BEGIN
   BB_G1.Konfig.Res_0 := FALSE;
   BB_G1.Konfig.Res_1 := FALSE;
   BB_G1.Konfig.Res_2 := FALSE;
   BB_G1.Konfig.Res_3 := FALSE;
   BB_G1.Konfig.Res_4 := FALSE;
   BB_G1.Konfig.Res_5 := FALSE;
   BB_G1.Konfig.Res_6 := FALSE;
   BB_G1.Konfig.Res_7 := FALSE;
   BB_G1.Konfig.Res_8 := FALSE;
   BB_G1.Konfig.Res_9 := FALSE;
   BB_G1.Konfig.Res_10 := FALSE;
   BB_G1.Konfig.Res_11 := FALSE;
   BB_G1.Konfig.Res_12 := FALSE;
   BB_G1.Konfig.Res_13 := FALSE;
   BB_G1.Konfig.Res_14 := FALSE;
   BB_G1.Konfig.Res_15 := FALSE;
   BB_G1.Konfig.Res_16 := FALSE;
   BB_G1.Konfig.Res_17 := FALSE;
   BB_G1.Konfig.Res_18 := FALSE;
   BB_G1.Konfig.Res_19 := FALSE;
   BB_G1.Konfig.Res_20 := FALSE;
   BB_G1.Konfig.Res_21 := FALSE;
   BB_G1.Konfig.Res_22 := FALSE;
   BB_G1.Konfig.Res_23 := FALSE;
   BB_G1.Konfig.Res_24 := FALSE;
   BB_G1.Konfig.Res_25 := FALSE;
   BB_G1.Konfig.Res_26 := FALSE;
   BB_G1.Konfig.Res_27 := FALSE;
   BB_G1.Konfig.Res_28 := FALSE;
   BB_G1.Konfig.Res_29 := FALSE;
   BB_G1.Konfig.Res_30 := FALSE;
   BB_G1.Konfig.Prm_Set := FALSE;
   BB_G1.P_nenn := 1.0;
   BB_G1.EZ_max := 0;
   BB_G1.AZ_min := 5;
   BB_G1.AZ_Rev := 10;
   BB_G1.VZ_St := 5;
   BB_G1.UeZ_Endl := 120;
   BB_G1.UeZ_BF := 120;
   BB_G1.Prio_NS := 0;
   BB_G1.Prio_ECS := 0;
   BB_G1.Prio_NA := 0;
   BB_G1.ESV_NA := 5;
   BB_G2.Konfig.Res_0 := FALSE;
   BB_G2.Konfig.Res_1 := FALSE;
   BB_G2.Konfig.Res_2 := FALSE;
   BB_G2.Konfig.Res_3 := FALSE;
   BB_G2.Konfig.Res_4 := FALSE;
   BB_G2.Konfig.Res_5 := FALSE;
   BB_G2.Konfig.Res_6 := FALSE;
   BB_G2.Konfig.Res_7 := FALSE;
   BB_G2.Konfig.Res_8 := FALSE;
   BB_G2.Konfig.Res_9 := FALSE;
   BB_G2.Konfig.Res_10 := FALSE;
   BB_G2.Konfig.Res_11 := FALSE;
   BB_G2.Konfig.Res_12 := FALSE;
   BB_G2.Konfig.Res_13 := FALSE;
   BB_G2.Konfig.Res_14 := FALSE;
   BB_G2.Konfig.Res_15 := FALSE;
   BB_G2.Konfig.Res_16 := FALSE;
   BB_G2.Konfig.Res_17 := FALSE;
   BB_G2.Konfig.Res_18 := FALSE;
   BB_G2.Konfig.Res_19 := FALSE;
   BB_G2.Konfig.Res_20 := FALSE;
   BB_G2.Konfig.Res_21 := FALSE;
   BB_G2.Konfig.Res_22 := FALSE;
   BB_G2.Konfig.Res_23 := FALSE;
   BB_G2.Konfig.Res_24 := FALSE;
   BB_G2.Konfig.Res_25 := FALSE;
   BB_G2.Konfig.Res_26 := FALSE;
   BB_G2.Konfig.Res_27 := FALSE;
   BB_G2.Konfig.Res_28 := FALSE;
   BB_G2.Konfig.Res_29 := FALSE;
   BB_G2.Konfig.Res_30 := FALSE;
   BB_G2.Konfig.Prm_Set := FALSE;
   BB_G2.P_nenn := 1.0;
   BB_G2.EZ_max := 0;
   BB_G2.AZ_min := 5;
   BB_G2.AZ_Rev := 10;
   BB_G2.VZ_St := 5;
   BB_G2.UeZ_Endl := 120;
   BB_G2.UeZ_BF := 15;
   BB_G2.Prio_NS := 0;
   BB_G2.Prio_ECS := 0;
   BB_G2.Prio_NA := 0;
   BB_G2.ESV_NA := 5;
   BB_G3.Konfig.Res_0 := FALSE;
   BB_G3.Konfig.Res_1 := FALSE;
   BB_G3.Konfig.Res_2 := FALSE;
   BB_G3.Konfig.Res_3 := FALSE;
   BB_G3.Konfig.Res_4 := FALSE;
   BB_G3.Konfig.Res_5 := FALSE;
   BB_G3.Konfig.Res_6 := FALSE;
   BB_G3.Konfig.Res_7 := FALSE;
   BB_G3.Konfig.Res_8 := FALSE;
   BB_G3.Konfig.Res_9 := FALSE;
   BB_G3.Konfig.Res_10 := FALSE;
   BB_G3.Konfig.Res_11 := FALSE;
   BB_G3.Konfig.Res_12 := FALSE;
   BB_G3.Konfig.Res_13 := FALSE;
   BB_G3.Konfig.Res_14 := FALSE;
   BB_G3.Konfig.Res_15 := FALSE;
   BB_G3.Konfig.Res_16 := FALSE;
   BB_G3.Konfig.Res_17 := FALSE;
   BB_G3.Konfig.Res_18 := FALSE;
   BB_G3.Konfig.Res_19 := FALSE;
   BB_G3.Konfig.Res_20 := FALSE;
   BB_G3.Konfig.Res_21 := FALSE;
   BB_G3.Konfig.Res_22 := FALSE;
   BB_G3.Konfig.Res_23 := FALSE;
   BB_G3.Konfig.Res_24 := FALSE;
   BB_G3.Konfig.Res_25 := FALSE;
   BB_G3.Konfig.Res_26 := FALSE;
   BB_G3.Konfig.Res_27 := FALSE;
   BB_G3.Konfig.Res_28 := FALSE;
   BB_G3.Konfig.Res_29 := FALSE;
   BB_G3.Konfig.Res_30 := FALSE;
   BB_G3.Konfig.Prm_Set := FALSE;
   BB_G3.P_nenn := 1.0;
   BB_G3.EZ_max := 0;
   BB_G3.AZ_min := 5;
   BB_G3.AZ_Rev := 10;
   BB_G3.VZ_St := 5;
   BB_G3.UeZ_Endl := 120;
   BB_G3.UeZ_BF := 15;
   BB_G3.Prio_NS := 0;
   BB_G3.Prio_ECS := 0;
   BB_G3.Prio_NA := 0;
   BB_G3.ESV_NA := 5;
   BB_SHL_G1.Konfig.Res_0 := FALSE;
   BB_SHL_G1.Konfig.Res_1 := FALSE;
   BB_SHL_G1.Konfig.Res_2 := FALSE;
   BB_SHL_G1.Konfig.Res_3 := FALSE;
   BB_SHL_G1.Konfig.Res_4 := FALSE;
   BB_SHL_G1.Konfig.Res_5 := FALSE;
   BB_SHL_G1.Konfig.Res_6 := FALSE;
   BB_SHL_G1.Konfig.Res_7 := FALSE;
   BB_SHL_G1.Konfig.Res_8 := FALSE;
   BB_SHL_G1.Konfig.Res_9 := FALSE;
   BB_SHL_G1.Konfig.Res_10 := FALSE;
   BB_SHL_G1.Konfig.Res_11 := FALSE;
   BB_SHL_G1.Konfig.Res_12 := FALSE;
   BB_SHL_G1.Konfig.Res_13 := FALSE;
   BB_SHL_G1.Konfig.Res_14 := FALSE;
   BB_SHL_G1.Konfig.Res_15 := FALSE;
   BB_SHL_G1.Konfig.Res_16 := FALSE;
   BB_SHL_G1.Konfig.Res_17 := FALSE;
   BB_SHL_G1.Konfig.Res_18 := FALSE;
   BB_SHL_G1.Konfig.Res_19 := FALSE;
   BB_SHL_G1.Konfig.Res_20 := FALSE;
   BB_SHL_G1.Konfig.Res_21 := FALSE;
   BB_SHL_G1.Konfig.Res_22 := FALSE;
   BB_SHL_G1.Konfig.Res_23 := FALSE;
   BB_SHL_G1.Konfig.Res_24 := FALSE;
   BB_SHL_G1.Konfig.Res_25 := FALSE;
   BB_SHL_G1.Konfig.Res_26 := FALSE;
   BB_SHL_G1.Konfig.Res_27 := FALSE;
   BB_SHL_G1.Konfig.Res_28 := FALSE;
   BB_SHL_G1.Konfig.Res_29 := FALSE;
   BB_SHL_G1.Konfig.Res_30 := FALSE;
   BB_SHL_G1.Konfig.Prm_Set := FALSE;
   BB_SHL_G1.P_nenn := 1.0;
   BB_SHL_G1.EZ_max := 0;
   BB_SHL_G1.AZ_min := 5;
   BB_SHL_G1.AZ_Rev := 10;
   BB_SHL_G1.VZ_St := 5;
   BB_SHL_G1.UeZ_Endl := 120;
   BB_SHL_G1.UeZ_BF := 15;
   BB_SHL_G1.Prio_NS := 0;
   BB_SHL_G1.Prio_ECS := 0;
   BB_SHL_G1.Prio_NA := 0;
   BB_SHL_G1.ESV_NA := 5;
   BB_SHL_G2.Konfig.Res_0 := FALSE;
   BB_SHL_G2.Konfig.Res_1 := FALSE;
   BB_SHL_G2.Konfig.Res_2 := FALSE;
   BB_SHL_G2.Konfig.Res_3 := FALSE;
   BB_SHL_G2.Konfig.Res_4 := FALSE;
   BB_SHL_G2.Konfig.Res_5 := FALSE;
   BB_SHL_G2.Konfig.Res_6 := FALSE;
   BB_SHL_G2.Konfig.Res_7 := FALSE;
   BB_SHL_G2.Konfig.Res_8 := FALSE;
   BB_SHL_G2.Konfig.Res_9 := FALSE;
   BB_SHL_G2.Konfig.Res_10 := FALSE;
   BB_SHL_G2.Konfig.Res_11 := FALSE;
   BB_SHL_G2.Konfig.Res_12 := FALSE;
   BB_SHL_G2.Konfig.Res_13 := FALSE;
   BB_SHL_G2.Konfig.Res_14 := FALSE;
   BB_SHL_G2.Konfig.Res_15 := FALSE;
   BB_SHL_G2.Konfig.Res_16 := FALSE;
   BB_SHL_G2.Konfig.Res_17 := FALSE;
   BB_SHL_G2.Konfig.Res_18 := FALSE;
   BB_SHL_G2.Konfig.Res_19 := FALSE;
   BB_SHL_G2.Konfig.Res_20 := FALSE;
   BB_SHL_G2.Konfig.Res_21 := FALSE;
   BB_SHL_G2.Konfig.Res_22 := FALSE;
   BB_SHL_G2.Konfig.Res_23 := FALSE;
   BB_SHL_G2.Konfig.Res_24 := FALSE;
   BB_SHL_G2.Konfig.Res_25 := FALSE;
   BB_SHL_G2.Konfig.Res_26 := FALSE;
   BB_SHL_G2.Konfig.Res_27 := FALSE;
   BB_SHL_G2.Konfig.Res_28 := FALSE;
   BB_SHL_G2.Konfig.Res_29 := FALSE;
   BB_SHL_G2.Konfig.Res_30 := FALSE;
   BB_SHL_G2.Konfig.Prm_Set := FALSE;
   BB_SHL_G2.P_nenn := 1.0;
   BB_SHL_G2.EZ_max := 0;
   BB_SHL_G2.AZ_min := 5;
   BB_SHL_G2.AZ_Rev := 10;
   BB_SHL_G2.VZ_St := 5;
   BB_SHL_G2.UeZ_Endl := 120;
   BB_SHL_G2.UeZ_BF := 15;
   BB_SHL_G2.Prio_NS := 0;
   BB_SHL_G2.Prio_ECS := 0;
   BB_SHL_G2.Prio_NA := 0;
   BB_SHL_G2.ESV_NA := 5;
   BB_SHL_G3.Konfig.Res_0 := FALSE;
   BB_SHL_G3.Konfig.Res_1 := FALSE;
   BB_SHL_G3.Konfig.Res_2 := FALSE;
   BB_SHL_G3.Konfig.Res_3 := FALSE;
   BB_SHL_G3.Konfig.Res_4 := FALSE;
   BB_SHL_G3.Konfig.Res_5 := FALSE;
   BB_SHL_G3.Konfig.Res_6 := FALSE;
   BB_SHL_G3.Konfig.Res_7 := FALSE;
   BB_SHL_G3.Konfig.Res_8 := FALSE;
   BB_SHL_G3.Konfig.Res_9 := FALSE;
   BB_SHL_G3.Konfig.Res_10 := FALSE;
   BB_SHL_G3.Konfig.Res_11 := FALSE;
   BB_SHL_G3.Konfig.Res_12 := FALSE;
   BB_SHL_G3.Konfig.Res_13 := FALSE;
   BB_SHL_G3.Konfig.Res_14 := FALSE;
   BB_SHL_G3.Konfig.Res_15 := FALSE;
   BB_SHL_G3.Konfig.Res_16 := FALSE;
   BB_SHL_G3.Konfig.Res_17 := FALSE;
   BB_SHL_G3.Konfig.Res_18 := FALSE;
   BB_SHL_G3.Konfig.Res_19 := FALSE;
   BB_SHL_G3.Konfig.Res_20 := FALSE;
   BB_SHL_G3.Konfig.Res_21 := FALSE;
   BB_SHL_G3.Konfig.Res_22 := FALSE;
   BB_SHL_G3.Konfig.Res_23 := FALSE;
   BB_SHL_G3.Konfig.Res_24 := FALSE;
   BB_SHL_G3.Konfig.Res_25 := FALSE;
   BB_SHL_G3.Konfig.Res_26 := FALSE;
   BB_SHL_G3.Konfig.Res_27 := FALSE;
   BB_SHL_G3.Konfig.Res_28 := FALSE;
   BB_SHL_G3.Konfig.Res_29 := FALSE;
   BB_SHL_G3.Konfig.Res_30 := FALSE;
   BB_SHL_G3.Konfig.Prm_Set := FALSE;
   BB_SHL_G3.P_nenn := 1.0;
   BB_SHL_G3.EZ_max := 0;
   BB_SHL_G3.AZ_min := 5;
   BB_SHL_G3.AZ_Rev := 10;
   BB_SHL_G3.VZ_St := 5;
   BB_SHL_G3.UeZ_Endl := 120;
   BB_SHL_G3.UeZ_BF := 15;
   BB_SHL_G3.Prio_NS := 0;
   BB_SHL_G3.Prio_ECS := 0;
   BB_SHL_G3.Prio_NA := 0;
   BB_SHL_G3.ESV_NA := 5;
   BB_AV.Konfig.Res_0 := FALSE;
   BB_AV.Konfig.Res_1 := FALSE;
   BB_AV.Konfig.Res_2 := FALSE;
   BB_AV.Konfig.Res_3 := FALSE;
   BB_AV.Konfig.Res_4 := FALSE;
   BB_AV.Konfig.Res_5 := FALSE;
   BB_AV.Konfig.Res_6 := FALSE;
   BB_AV.Konfig.Res_7 := FALSE;
   BB_AV.Konfig.Res_8 := FALSE;
   BB_AV.Konfig.Res_9 := FALSE;
   BB_AV.Konfig.Res_10 := FALSE;
   BB_AV.Konfig.Res_11 := FALSE;
   BB_AV.Konfig.Res_12 := FALSE;
   BB_AV.Konfig.Res_13 := FALSE;
   BB_AV.Konfig.Res_14 := FALSE;
   BB_AV.Konfig.Res_15 := FALSE;
   BB_AV.Konfig.Res_16 := FALSE;
   BB_AV.Konfig.Res_17 := FALSE;
   BB_AV.Konfig.Res_18 := FALSE;
   BB_AV.Konfig.Res_19 := FALSE;
   BB_AV.Konfig.Res_20 := FALSE;
   BB_AV.Konfig.Res_21 := FALSE;
   BB_AV.Konfig.Res_22 := FALSE;
   BB_AV.Konfig.Res_23 := FALSE;
   BB_AV.Konfig.Res_24 := FALSE;
   BB_AV.Konfig.Res_25 := FALSE;
   BB_AV.Konfig.Res_26 := FALSE;
   BB_AV.Konfig.Res_27 := FALSE;
   BB_AV.Konfig.Res_28 := FALSE;
   BB_AV.Konfig.Res_29 := FALSE;
   BB_AV.Konfig.Res_30 := FALSE;
   BB_AV.Konfig.Prm_Set := FALSE;
   BB_AV.P_nenn := 1.0;
   BB_AV.EZ_max := 0;
   BB_AV.AZ_min := 5;
   BB_AV.AZ_Rev := 10;
   BB_AV.VZ_St := 5;
   BB_AV.UeZ_Endl := 120;
   BB_AV.UeZ_BF := 15;
   BB_AV.Prio_NS := 0;
   BB_AV.Prio_ECS := 0;
   BB_AV.Prio_NA := 0;
   BB_AV.ESV_NA := 5;
   BB_LS1.Konfig.Res_0 := FALSE;
   BB_LS1.Konfig.Res_1 := FALSE;
   BB_LS1.Konfig.Res_2 := FALSE;
   BB_LS1.Konfig.Res_3 := FALSE;
   BB_LS1.Konfig.Res_4 := FALSE;
   BB_LS1.Konfig.Res_5 := FALSE;
   BB_LS1.Konfig.Res_6 := FALSE;
   BB_LS1.Konfig.Res_7 := FALSE;
   BB_LS1.Konfig.Res_8 := FALSE;
   BB_LS1.Konfig.Res_9 := FALSE;
   BB_LS1.Konfig.Res_10 := FALSE;
   BB_LS1.Konfig.Res_11 := FALSE;
   BB_LS1.Konfig.Res_12 := FALSE;
   BB_LS1.Konfig.Res_13 := FALSE;
   BB_LS1.Konfig.Res_14 := FALSE;
   BB_LS1.Konfig.Res_15 := FALSE;
   BB_LS1.Konfig.Res_16 := FALSE;
   BB_LS1.Konfig.Res_17 := FALSE;
   BB_LS1.Konfig.Res_18 := FALSE;
   BB_LS1.Konfig.Res_19 := FALSE;
   BB_LS1.Konfig.Res_20 := FALSE;
   BB_LS1.Konfig.Res_21 := FALSE;
   BB_LS1.Konfig.Res_22 := FALSE;
   BB_LS1.Konfig.Res_23 := FALSE;
   BB_LS1.Konfig.Res_24 := FALSE;
   BB_LS1.Konfig.Res_25 := FALSE;
   BB_LS1.Konfig.Res_26 := FALSE;
   BB_LS1.Konfig.Res_27 := FALSE;
   BB_LS1.Konfig.Res_28 := FALSE;
   BB_LS1.Konfig.Res_29 := FALSE;
   BB_LS1.Konfig.Res_30 := FALSE;
   BB_LS1.Konfig.Prm_Set := FALSE;
   BB_LS1.P_nenn := 1.0;
   BB_LS1.EZ_max := 0;
   BB_LS1.AZ_min := 5;
   BB_LS1.AZ_Rev := 10;
   BB_LS1.VZ_St := 5;
   BB_LS1.UeZ_Endl := 120;
   BB_LS1.UeZ_BF := 15;
   BB_LS1.Prio_NS := 0;
   BB_LS1.Prio_ECS := 0;
   BB_LS1.Prio_NA := 0;
   BB_LS1.ESV_NA := 5;
   BB_LS2.Konfig.Res_0 := FALSE;
   BB_LS2.Konfig.Res_1 := FALSE;
   BB_LS2.Konfig.Res_2 := FALSE;
   BB_LS2.Konfig.Res_3 := FALSE;
   BB_LS2.Konfig.Res_4 := FALSE;
   BB_LS2.Konfig.Res_5 := FALSE;
   BB_LS2.Konfig.Res_6 := FALSE;
   BB_LS2.Konfig.Res_7 := FALSE;
   BB_LS2.Konfig.Res_8 := FALSE;
   BB_LS2.Konfig.Res_9 := FALSE;
   BB_LS2.Konfig.Res_10 := FALSE;
   BB_LS2.Konfig.Res_11 := FALSE;
   BB_LS2.Konfig.Res_12 := FALSE;
   BB_LS2.Konfig.Res_13 := FALSE;
   BB_LS2.Konfig.Res_14 := FALSE;
   BB_LS2.Konfig.Res_15 := FALSE;
   BB_LS2.Konfig.Res_16 := FALSE;
   BB_LS2.Konfig.Res_17 := FALSE;
   BB_LS2.Konfig.Res_18 := FALSE;
   BB_LS2.Konfig.Res_19 := FALSE;
   BB_LS2.Konfig.Res_20 := FALSE;
   BB_LS2.Konfig.Res_21 := FALSE;
   BB_LS2.Konfig.Res_22 := FALSE;
   BB_LS2.Konfig.Res_23 := FALSE;
   BB_LS2.Konfig.Res_24 := FALSE;
   BB_LS2.Konfig.Res_25 := FALSE;
   BB_LS2.Konfig.Res_26 := FALSE;
   BB_LS2.Konfig.Res_27 := FALSE;
   BB_LS2.Konfig.Res_28 := FALSE;
   BB_LS2.Konfig.Res_29 := FALSE;
   BB_LS2.Konfig.Res_30 := FALSE;
   BB_LS2.Konfig.Prm_Set := FALSE;
   BB_LS2.P_nenn := 1.0;
   BB_LS2.EZ_max := 0;
   BB_LS2.AZ_min := 5;
   BB_LS2.AZ_Rev := 10;
   BB_LS2.VZ_St := 5;
   BB_LS2.UeZ_Endl := 120;
   BB_LS2.UeZ_BF := 15;
   BB_LS2.Prio_NS := 0;
   BB_LS2.Prio_ECS := 0;
   BB_LS2.Prio_NA := 0;
   BB_LS2.ESV_NA := 5;
   BB1_RZP1.Konfig.Res_0 := FALSE;
   BB1_RZP1.Konfig.Res_1 := FALSE;
   BB1_RZP1.Konfig.Res_2 := FALSE;
   BB1_RZP1.Konfig.Res_3 := FALSE;
   BB1_RZP1.Konfig.Res_4 := FALSE;
   BB1_RZP1.Konfig.Res_5 := FALSE;
   BB1_RZP1.Konfig.Res_6 := FALSE;
   BB1_RZP1.Konfig.Res_7 := FALSE;
   BB1_RZP1.Konfig.Res_8 := FALSE;
   BB1_RZP1.Konfig.Res_9 := FALSE;
   BB1_RZP1.Konfig.Res_10 := FALSE;
   BB1_RZP1.Konfig.Res_11 := FALSE;
   BB1_RZP1.Konfig.Res_12 := FALSE;
   BB1_RZP1.Konfig.Res_13 := FALSE;
   BB1_RZP1.Konfig.Res_14 := FALSE;
   BB1_RZP1.Konfig.Res_15 := FALSE;
   BB1_RZP1.Konfig.Res_16 := FALSE;
   BB1_RZP1.Konfig.Res_17 := FALSE;
   BB1_RZP1.Konfig.Res_18 := FALSE;
   BB1_RZP1.Konfig.Res_19 := FALSE;
   BB1_RZP1.Konfig.Res_20 := FALSE;
   BB1_RZP1.Konfig.Res_21 := FALSE;
   BB1_RZP1.Konfig.Res_22 := FALSE;
   BB1_RZP1.Konfig.Res_23 := FALSE;
   BB1_RZP1.Konfig.Res_24 := FALSE;
   BB1_RZP1.Konfig.Res_25 := FALSE;
   BB1_RZP1.Konfig.Res_26 := FALSE;
   BB1_RZP1.Konfig.Res_27 := FALSE;
   BB1_RZP1.Konfig.Res_28 := FALSE;
   BB1_RZP1.Konfig.Res_29 := FALSE;
   BB1_RZP1.Konfig.Res_30 := FALSE;
   BB1_RZP1.Konfig.Prm_Set := FALSE;
   BB1_RZP1.P_nenn := 2.0;
   BB1_RZP1.EZ_max := 0;
   BB1_RZP1.AZ_min := 5;
   BB1_RZP1.AZ_Rev := 10;
   BB1_RZP1.VZ_St := 5;
   BB1_RZP1.UeZ_Endl := 300;
   BB1_RZP1.UeZ_BF := 15;
   BB1_RZP1.Prio_NS := 0;
   BB1_RZP1.Prio_ECS := 0;
   BB1_RZP1.Prio_NA := 0;
   BB1_RZP1.ESV_NA := 5;
   BB1_RZP2.Konfig.Res_0 := FALSE;
   BB1_RZP2.Konfig.Res_1 := FALSE;
   BB1_RZP2.Konfig.Res_2 := FALSE;
   BB1_RZP2.Konfig.Res_3 := FALSE;
   BB1_RZP2.Konfig.Res_4 := FALSE;
   BB1_RZP2.Konfig.Res_5 := FALSE;
   BB1_RZP2.Konfig.Res_6 := FALSE;
   BB1_RZP2.Konfig.Res_7 := FALSE;
   BB1_RZP2.Konfig.Res_8 := FALSE;
   BB1_RZP2.Konfig.Res_9 := FALSE;
   BB1_RZP2.Konfig.Res_10 := FALSE;
   BB1_RZP2.Konfig.Res_11 := FALSE;
   BB1_RZP2.Konfig.Res_12 := FALSE;
   BB1_RZP2.Konfig.Res_13 := FALSE;
   BB1_RZP2.Konfig.Res_14 := FALSE;
   BB1_RZP2.Konfig.Res_15 := FALSE;
   BB1_RZP2.Konfig.Res_16 := FALSE;
   BB1_RZP2.Konfig.Res_17 := FALSE;
   BB1_RZP2.Konfig.Res_18 := FALSE;
   BB1_RZP2.Konfig.Res_19 := FALSE;
   BB1_RZP2.Konfig.Res_20 := FALSE;
   BB1_RZP2.Konfig.Res_21 := FALSE;
   BB1_RZP2.Konfig.Res_22 := FALSE;
   BB1_RZP2.Konfig.Res_23 := FALSE;
   BB1_RZP2.Konfig.Res_24 := FALSE;
   BB1_RZP2.Konfig.Res_25 := FALSE;
   BB1_RZP2.Konfig.Res_26 := FALSE;
   BB1_RZP2.Konfig.Res_27 := FALSE;
   BB1_RZP2.Konfig.Res_28 := FALSE;
   BB1_RZP2.Konfig.Res_29 := FALSE;
   BB1_RZP2.Konfig.Res_30 := FALSE;
   BB1_RZP2.Konfig.Prm_Set := FALSE;
   BB1_RZP2.P_nenn := 1.0;
   BB1_RZP2.EZ_max := 0;
   BB1_RZP2.AZ_min := 5;
   BB1_RZP2.AZ_Rev := 10;
   BB1_RZP2.VZ_St := 5;
   BB1_RZP2.UeZ_Endl := 120;
   BB1_RZP2.UeZ_BF := 15;
   BB1_RZP2.Prio_NS := 0;
   BB1_RZP2.Prio_ECS := 0;
   BB1_RZP2.Prio_NA := 0;
   BB1_RZP2.ESV_NA := 5;
   BB1_UeSP.Konfig.Res_0 := FALSE;
   BB1_UeSP.Konfig.Res_1 := FALSE;
   BB1_UeSP.Konfig.Res_2 := FALSE;
   BB1_UeSP.Konfig.Res_3 := FALSE;
   BB1_UeSP.Konfig.Res_4 := FALSE;
   BB1_UeSP.Konfig.Res_5 := FALSE;
   BB1_UeSP.Konfig.Res_6 := FALSE;
   BB1_UeSP.Konfig.Res_7 := FALSE;
   BB1_UeSP.Konfig.Res_8 := FALSE;
   BB1_UeSP.Konfig.Res_9 := FALSE;
   BB1_UeSP.Konfig.Res_10 := FALSE;
   BB1_UeSP.Konfig.Res_11 := FALSE;
   BB1_UeSP.Konfig.Res_12 := FALSE;
   BB1_UeSP.Konfig.Res_13 := FALSE;
   BB1_UeSP.Konfig.Res_14 := FALSE;
   BB1_UeSP.Konfig.Res_15 := FALSE;
   BB1_UeSP.Konfig.Res_16 := FALSE;
   BB1_UeSP.Konfig.Res_17 := FALSE;
   BB1_UeSP.Konfig.Res_18 := FALSE;
   BB1_UeSP.Konfig.Res_19 := FALSE;
   BB1_UeSP.Konfig.Res_20 := FALSE;
   BB1_UeSP.Konfig.Res_21 := FALSE;
   BB1_UeSP.Konfig.Res_22 := FALSE;
   BB1_UeSP.Konfig.Res_23 := FALSE;
   BB1_UeSP.Konfig.Res_24 := FALSE;
   BB1_UeSP.Konfig.Res_25 := FALSE;
   BB1_UeSP.Konfig.Res_26 := FALSE;
   BB1_UeSP.Konfig.Res_27 := FALSE;
   BB1_UeSP.Konfig.Res_28 := FALSE;
   BB1_UeSP.Konfig.Res_29 := FALSE;
   BB1_UeSP.Konfig.Res_30 := FALSE;
   BB1_UeSP.Konfig.Prm_Set := FALSE;
   BB1_UeSP.P_nenn := 1.0;
   BB1_UeSP.EZ_max := 0;
   BB1_UeSP.AZ_min := 5;
   BB1_UeSP.AZ_Rev := 10;
   BB1_UeSP.VZ_St := 5;
   BB1_UeSP.UeZ_Endl := 120;
   BB1_UeSP.UeZ_BF := 15;
   BB1_UeSP.Prio_NS := 0;
   BB1_UeSP.Prio_ECS := 0;
   BB1_UeSP.Prio_NA := 0;
   BB1_UeSP.ESV_NA := 5;
   BB1_AS1.Konfig.Res_0 := FALSE;
   BB1_AS1.Konfig.Res_1 := FALSE;
   BB1_AS1.Konfig.Res_2 := FALSE;
   BB1_AS1.Konfig.Res_3 := FALSE;
   BB1_AS1.Konfig.Res_4 := FALSE;
   BB1_AS1.Konfig.Res_5 := FALSE;
   BB1_AS1.Konfig.Res_6 := FALSE;
   BB1_AS1.Konfig.Res_7 := FALSE;
   BB1_AS1.Konfig.Res_8 := FALSE;
   BB1_AS1.Konfig.Res_9 := FALSE;
   BB1_AS1.Konfig.Res_10 := FALSE;
   BB1_AS1.Konfig.Res_11 := FALSE;
   BB1_AS1.Konfig.Res_12 := FALSE;
   BB1_AS1.Konfig.Res_13 := FALSE;
   BB1_AS1.Konfig.Res_14 := FALSE;
   BB1_AS1.Konfig.Res_15 := FALSE;
   BB1_AS1.Konfig.Res_16 := FALSE;
   BB1_AS1.Konfig.Res_17 := FALSE;
   BB1_AS1.Konfig.Res_18 := FALSE;
   BB1_AS1.Konfig.Res_19 := FALSE;
   BB1_AS1.Konfig.Res_20 := FALSE;
   BB1_AS1.Konfig.Res_21 := FALSE;
   BB1_AS1.Konfig.Res_22 := FALSE;
   BB1_AS1.Konfig.Res_23 := FALSE;
   BB1_AS1.Konfig.Res_24 := FALSE;
   BB1_AS1.Konfig.Res_25 := FALSE;
   BB1_AS1.Konfig.Res_26 := FALSE;
   BB1_AS1.Konfig.Res_27 := FALSE;
   BB1_AS1.Konfig.Res_28 := FALSE;
   BB1_AS1.Konfig.Res_29 := FALSE;
   BB1_AS1.Konfig.Res_30 := FALSE;
   BB1_AS1.Konfig.Prm_Set := FALSE;
   BB1_AS1.P_nenn := 1.0;
   BB1_AS1.EZ_max := 0;
   BB1_AS1.AZ_min := 5;
   BB1_AS1.AZ_Rev := 10;
   BB1_AS1.VZ_St := 5;
   BB1_AS1.UeZ_Endl := 120;
   BB1_AS1.UeZ_BF := 15;
   BB1_AS1.Prio_NS := 0;
   BB1_AS1.Prio_ECS := 0;
   BB1_AS1.Prio_NA := 0;
   BB1_AS1.ESV_NA := 5;
   BB1_AS2.Konfig.Res_0 := FALSE;
   BB1_AS2.Konfig.Res_1 := FALSE;
   BB1_AS2.Konfig.Res_2 := FALSE;
   BB1_AS2.Konfig.Res_3 := FALSE;
   BB1_AS2.Konfig.Res_4 := FALSE;
   BB1_AS2.Konfig.Res_5 := FALSE;
   BB1_AS2.Konfig.Res_6 := FALSE;
   BB1_AS2.Konfig.Res_7 := FALSE;
   BB1_AS2.Konfig.Res_8 := FALSE;
   BB1_AS2.Konfig.Res_9 := FALSE;
   BB1_AS2.Konfig.Res_10 := FALSE;
   BB1_AS2.Konfig.Res_11 := FALSE;
   BB1_AS2.Konfig.Res_12 := FALSE;
   BB1_AS2.Konfig.Res_13 := FALSE;
   BB1_AS2.Konfig.Res_14 := FALSE;
   BB1_AS2.Konfig.Res_15 := FALSE;
   BB1_AS2.Konfig.Res_16 := FALSE;
   BB1_AS2.Konfig.Res_17 := FALSE;
   BB1_AS2.Konfig.Res_18 := FALSE;
   BB1_AS2.Konfig.Res_19 := FALSE;
   BB1_AS2.Konfig.Res_20 := FALSE;
   BB1_AS2.Konfig.Res_21 := FALSE;
   BB1_AS2.Konfig.Res_22 := FALSE;
   BB1_AS2.Konfig.Res_23 := FALSE;
   BB1_AS2.Konfig.Res_24 := FALSE;
   BB1_AS2.Konfig.Res_25 := FALSE;
   BB1_AS2.Konfig.Res_26 := FALSE;
   BB1_AS2.Konfig.Res_27 := FALSE;
   BB1_AS2.Konfig.Res_28 := FALSE;
   BB1_AS2.Konfig.Res_29 := FALSE;
   BB1_AS2.Konfig.Res_30 := FALSE;
   BB1_AS2.Konfig.Prm_Set := FALSE;
   BB1_AS2.P_nenn := 1.0;
   BB1_AS2.EZ_max := 0;
   BB1_AS2.AZ_min := 5;
   BB1_AS2.AZ_Rev := 10;
   BB1_AS2.VZ_St := 5;
   BB1_AS2.UeZ_Endl := 120;
   BB1_AS2.UeZ_BF := 15;
   BB1_AS2.Prio_NS := 0;
   BB1_AS2.Prio_ECS := 0;
   BB1_AS2.Prio_NA := 0;
   BB1_AS2.ESV_NA := 5;
   BB1_SR1.Konfig.Res_0 := FALSE;
   BB1_SR1.Konfig.Res_1 := FALSE;
   BB1_SR1.Konfig.Res_2 := FALSE;
   BB1_SR1.Konfig.Res_3 := FALSE;
   BB1_SR1.Konfig.Res_4 := FALSE;
   BB1_SR1.Konfig.Res_5 := FALSE;
   BB1_SR1.Konfig.Res_6 := FALSE;
   BB1_SR1.Konfig.Res_7 := FALSE;
   BB1_SR1.Konfig.Res_8 := FALSE;
   BB1_SR1.Konfig.Res_9 := FALSE;
   BB1_SR1.Konfig.Res_10 := FALSE;
   BB1_SR1.Konfig.Res_11 := FALSE;
   BB1_SR1.Konfig.Res_12 := FALSE;
   BB1_SR1.Konfig.Res_13 := FALSE;
   BB1_SR1.Konfig.Res_14 := FALSE;
   BB1_SR1.Konfig.Res_15 := FALSE;
   BB1_SR1.Konfig.Res_16 := FALSE;
   BB1_SR1.Konfig.Res_17 := FALSE;
   BB1_SR1.Konfig.Res_18 := FALSE;
   BB1_SR1.Konfig.Res_19 := FALSE;
   BB1_SR1.Konfig.Res_20 := FALSE;
   BB1_SR1.Konfig.Res_21 := FALSE;
   BB1_SR1.Konfig.Res_22 := FALSE;
   BB1_SR1.Konfig.Res_23 := FALSE;
   BB1_SR1.Konfig.Res_24 := FALSE;
   BB1_SR1.Konfig.Res_25 := FALSE;
   BB1_SR1.Konfig.Res_26 := FALSE;
   BB1_SR1.Konfig.Res_27 := FALSE;
   BB1_SR1.Konfig.Res_28 := FALSE;
   BB1_SR1.Konfig.Res_29 := FALSE;
   BB1_SR1.Konfig.Res_30 := FALSE;
   BB1_SR1.Konfig.Prm_Set := FALSE;
   BB1_SR1.P_nenn := 1.0;
   BB1_SR1.EZ_max := 0;
   BB1_SR1.AZ_min := 5;
   BB1_SR1.AZ_Rev := 10;
   BB1_SR1.VZ_St := 5;
   BB1_SR1.UeZ_Endl := 120;
   BB1_SR1.UeZ_BF := 15;
   BB1_SR1.Prio_NS := 0;
   BB1_SR1.Prio_ECS := 0;
   BB1_SR1.Prio_NA := 0;
   BB1_SR1.ESV_NA := 5;
   BB1_SR2.Konfig.Res_0 := FALSE;
   BB1_SR2.Konfig.Res_1 := FALSE;
   BB1_SR2.Konfig.Res_2 := FALSE;
   BB1_SR2.Konfig.Res_3 := FALSE;
   BB1_SR2.Konfig.Res_4 := FALSE;
   BB1_SR2.Konfig.Res_5 := FALSE;
   BB1_SR2.Konfig.Res_6 := FALSE;
   BB1_SR2.Konfig.Res_7 := FALSE;
   BB1_SR2.Konfig.Res_8 := FALSE;
   BB1_SR2.Konfig.Res_9 := FALSE;
   BB1_SR2.Konfig.Res_10 := FALSE;
   BB1_SR2.Konfig.Res_11 := FALSE;
   BB1_SR2.Konfig.Res_12 := FALSE;
   BB1_SR2.Konfig.Res_13 := FALSE;
   BB1_SR2.Konfig.Res_14 := FALSE;
   BB1_SR2.Konfig.Res_15 := FALSE;
   BB1_SR2.Konfig.Res_16 := FALSE;
   BB1_SR2.Konfig.Res_17 := FALSE;
   BB1_SR2.Konfig.Res_18 := FALSE;
   BB1_SR2.Konfig.Res_19 := FALSE;
   BB1_SR2.Konfig.Res_20 := FALSE;
   BB1_SR2.Konfig.Res_21 := FALSE;
   BB1_SR2.Konfig.Res_22 := FALSE;
   BB1_SR2.Konfig.Res_23 := FALSE;
   BB1_SR2.Konfig.Res_24 := FALSE;
   BB1_SR2.Konfig.Res_25 := FALSE;
   BB1_SR2.Konfig.Res_26 := FALSE;
   BB1_SR2.Konfig.Res_27 := FALSE;
   BB1_SR2.Konfig.Res_28 := FALSE;
   BB1_SR2.Konfig.Res_29 := FALSE;
   BB1_SR2.Konfig.Res_30 := FALSE;
   BB1_SR2.Konfig.Prm_Set := FALSE;
   BB1_SR2.P_nenn := 1.0;
   BB1_SR2.EZ_max := 0;
   BB1_SR2.AZ_min := 5;
   BB1_SR2.AZ_Rev := 10;
   BB1_SR2.VZ_St := 5;
   BB1_SR2.UeZ_Endl := 120;
   BB1_SR2.UeZ_BF := 15;
   BB1_SR2.Prio_NS := 0;
   BB1_SR2.Prio_ECS := 0;
   BB1_SR2.Prio_NA := 0;
   BB1_SR2.ESV_NA := 5;
   BB2_RZP1.Konfig.Res_0 := FALSE;
   BB2_RZP1.Konfig.Res_1 := FALSE;
   BB2_RZP1.Konfig.Res_2 := FALSE;
   BB2_RZP1.Konfig.Res_3 := FALSE;
   BB2_RZP1.Konfig.Res_4 := FALSE;
   BB2_RZP1.Konfig.Res_5 := FALSE;
   BB2_RZP1.Konfig.Res_6 := FALSE;
   BB2_RZP1.Konfig.Res_7 := FALSE;
   BB2_RZP1.Konfig.Res_8 := FALSE;
   BB2_RZP1.Konfig.Res_9 := FALSE;
   BB2_RZP1.Konfig.Res_10 := FALSE;
   BB2_RZP1.Konfig.Res_11 := FALSE;
   BB2_RZP1.Konfig.Res_12 := FALSE;
   BB2_RZP1.Konfig.Res_13 := FALSE;
   BB2_RZP1.Konfig.Res_14 := FALSE;
   BB2_RZP1.Konfig.Res_15 := FALSE;
   BB2_RZP1.Konfig.Res_16 := FALSE;
   BB2_RZP1.Konfig.Res_17 := FALSE;
   BB2_RZP1.Konfig.Res_18 := FALSE;
   BB2_RZP1.Konfig.Res_19 := FALSE;
   BB2_RZP1.Konfig.Res_20 := FALSE;
   BB2_RZP1.Konfig.Res_21 := FALSE;
   BB2_RZP1.Konfig.Res_22 := FALSE;
   BB2_RZP1.Konfig.Res_23 := FALSE;
   BB2_RZP1.Konfig.Res_24 := FALSE;
   BB2_RZP1.Konfig.Res_25 := FALSE;
   BB2_RZP1.Konfig.Res_26 := FALSE;
   BB2_RZP1.Konfig.Res_27 := FALSE;
   BB2_RZP1.Konfig.Res_28 := FALSE;
   BB2_RZP1.Konfig.Res_29 := FALSE;
   BB2_RZP1.Konfig.Res_30 := FALSE;
   BB2_RZP1.Konfig.Prm_Set := FALSE;
   BB2_RZP1.P_nenn := 1.0;
   BB2_RZP1.EZ_max := 0;
   BB2_RZP1.AZ_min := 5;
   BB2_RZP1.AZ_Rev := 10;
   BB2_RZP1.VZ_St := 5;
   BB2_RZP1.UeZ_Endl := 120;
   BB2_RZP1.UeZ_BF := 15;
   BB2_RZP1.Prio_NS := 0;
   BB2_RZP1.Prio_ECS := 0;
   BB2_RZP1.Prio_NA := 0;
   BB2_RZP1.ESV_NA := 5;
   BB2_RZP2.Konfig.Res_0 := FALSE;
   BB2_RZP2.Konfig.Res_1 := FALSE;
   BB2_RZP2.Konfig.Res_2 := FALSE;
   BB2_RZP2.Konfig.Res_3 := FALSE;
   BB2_RZP2.Konfig.Res_4 := FALSE;
   BB2_RZP2.Konfig.Res_5 := FALSE;
   BB2_RZP2.Konfig.Res_6 := FALSE;
   BB2_RZP2.Konfig.Res_7 := FALSE;
   BB2_RZP2.Konfig.Res_8 := FALSE;
   BB2_RZP2.Konfig.Res_9 := FALSE;
   BB2_RZP2.Konfig.Res_10 := FALSE;
   BB2_RZP2.Konfig.Res_11 := FALSE;
   BB2_RZP2.Konfig.Res_12 := FALSE;
   BB2_RZP2.Konfig.Res_13 := FALSE;
   BB2_RZP2.Konfig.Res_14 := FALSE;
   BB2_RZP2.Konfig.Res_15 := FALSE;
   BB2_RZP2.Konfig.Res_16 := FALSE;
   BB2_RZP2.Konfig.Res_17 := FALSE;
   BB2_RZP2.Konfig.Res_18 := FALSE;
   BB2_RZP2.Konfig.Res_19 := FALSE;
   BB2_RZP2.Konfig.Res_20 := FALSE;
   BB2_RZP2.Konfig.Res_21 := FALSE;
   BB2_RZP2.Konfig.Res_22 := FALSE;
   BB2_RZP2.Konfig.Res_23 := FALSE;
   BB2_RZP2.Konfig.Res_24 := FALSE;
   BB2_RZP2.Konfig.Res_25 := FALSE;
   BB2_RZP2.Konfig.Res_26 := FALSE;
   BB2_RZP2.Konfig.Res_27 := FALSE;
   BB2_RZP2.Konfig.Res_28 := FALSE;
   BB2_RZP2.Konfig.Res_29 := FALSE;
   BB2_RZP2.Konfig.Res_30 := FALSE;
   BB2_RZP2.Konfig.Prm_Set := FALSE;
   BB2_RZP2.P_nenn := 1.0;
   BB2_RZP2.EZ_max := 0;
   BB2_RZP2.AZ_min := 5;
   BB2_RZP2.AZ_Rev := 10;
   BB2_RZP2.VZ_St := 5;
   BB2_RZP2.UeZ_Endl := 120;
   BB2_RZP2.UeZ_BF := 15;
   BB2_RZP2.Prio_NS := 0;
   BB2_RZP2.Prio_ECS := 0;
   BB2_RZP2.Prio_NA := 0;
   BB2_RZP2.ESV_NA := 5;
   BB2_UeSP.Konfig.Res_0 := FALSE;
   BB2_UeSP.Konfig.Res_1 := FALSE;
   BB2_UeSP.Konfig.Res_2 := FALSE;
   BB2_UeSP.Konfig.Res_3 := FALSE;
   BB2_UeSP.Konfig.Res_4 := FALSE;
   BB2_UeSP.Konfig.Res_5 := FALSE;
   BB2_UeSP.Konfig.Res_6 := FALSE;
   BB2_UeSP.Konfig.Res_7 := FALSE;
   BB2_UeSP.Konfig.Res_8 := FALSE;
   BB2_UeSP.Konfig.Res_9 := FALSE;
   BB2_UeSP.Konfig.Res_10 := FALSE;
   BB2_UeSP.Konfig.Res_11 := FALSE;
   BB2_UeSP.Konfig.Res_12 := FALSE;
   BB2_UeSP.Konfig.Res_13 := FALSE;
   BB2_UeSP.Konfig.Res_14 := FALSE;
   BB2_UeSP.Konfig.Res_15 := FALSE;
   BB2_UeSP.Konfig.Res_16 := FALSE;
   BB2_UeSP.Konfig.Res_17 := FALSE;
   BB2_UeSP.Konfig.Res_18 := FALSE;
   BB2_UeSP.Konfig.Res_19 := FALSE;
   BB2_UeSP.Konfig.Res_20 := FALSE;
   BB2_UeSP.Konfig.Res_21 := FALSE;
   BB2_UeSP.Konfig.Res_22 := FALSE;
   BB2_UeSP.Konfig.Res_23 := FALSE;
   BB2_UeSP.Konfig.Res_24 := FALSE;
   BB2_UeSP.Konfig.Res_25 := FALSE;
   BB2_UeSP.Konfig.Res_26 := FALSE;
   BB2_UeSP.Konfig.Res_27 := FALSE;
   BB2_UeSP.Konfig.Res_28 := FALSE;
   BB2_UeSP.Konfig.Res_29 := FALSE;
   BB2_UeSP.Konfig.Res_30 := FALSE;
   BB2_UeSP.Konfig.Prm_Set := FALSE;
   BB2_UeSP.P_nenn := 1.0;
   BB2_UeSP.EZ_max := 0;
   BB2_UeSP.AZ_min := 5;
   BB2_UeSP.AZ_Rev := 10;
   BB2_UeSP.VZ_St := 5;
   BB2_UeSP.UeZ_Endl := 120;
   BB2_UeSP.UeZ_BF := 15;
   BB2_UeSP.Prio_NS := 0;
   BB2_UeSP.Prio_ECS := 0;
   BB2_UeSP.Prio_NA := 0;
   BB2_UeSP.ESV_NA := 5;
   BB2_AS1.Konfig.Res_0 := FALSE;
   BB2_AS1.Konfig.Res_1 := FALSE;
   BB2_AS1.Konfig.Res_2 := FALSE;
   BB2_AS1.Konfig.Res_3 := FALSE;
   BB2_AS1.Konfig.Res_4 := FALSE;
   BB2_AS1.Konfig.Res_5 := FALSE;
   BB2_AS1.Konfig.Res_6 := FALSE;
   BB2_AS1.Konfig.Res_7 := FALSE;
   BB2_AS1.Konfig.Res_8 := FALSE;
   BB2_AS1.Konfig.Res_9 := FALSE;
   BB2_AS1.Konfig.Res_10 := FALSE;
   BB2_AS1.Konfig.Res_11 := FALSE;
   BB2_AS1.Konfig.Res_12 := FALSE;
   BB2_AS1.Konfig.Res_13 := FALSE;
   BB2_AS1.Konfig.Res_14 := FALSE;
   BB2_AS1.Konfig.Res_15 := FALSE;
   BB2_AS1.Konfig.Res_16 := FALSE;
   BB2_AS1.Konfig.Res_17 := FALSE;
   BB2_AS1.Konfig.Res_18 := FALSE;
   BB2_AS1.Konfig.Res_19 := FALSE;
   BB2_AS1.Konfig.Res_20 := FALSE;
   BB2_AS1.Konfig.Res_21 := FALSE;
   BB2_AS1.Konfig.Res_22 := FALSE;
   BB2_AS1.Konfig.Res_23 := FALSE;
   BB2_AS1.Konfig.Res_24 := FALSE;
   BB2_AS1.Konfig.Res_25 := FALSE;
   BB2_AS1.Konfig.Res_26 := FALSE;
   BB2_AS1.Konfig.Res_27 := FALSE;
   BB2_AS1.Konfig.Res_28 := FALSE;
   BB2_AS1.Konfig.Res_29 := FALSE;
   BB2_AS1.Konfig.Res_30 := FALSE;
   BB2_AS1.Konfig.Prm_Set := FALSE;
   BB2_AS1.P_nenn := 1.0;
   BB2_AS1.EZ_max := 0;
   BB2_AS1.AZ_min := 5;
   BB2_AS1.AZ_Rev := 10;
   BB2_AS1.VZ_St := 5;
   BB2_AS1.UeZ_Endl := 120;
   BB2_AS1.UeZ_BF := 15;
   BB2_AS1.Prio_NS := 0;
   BB2_AS1.Prio_ECS := 0;
   BB2_AS1.Prio_NA := 0;
   BB2_AS1.ESV_NA := 5;
   BB2_AS2.Konfig.Res_0 := FALSE;
   BB2_AS2.Konfig.Res_1 := FALSE;
   BB2_AS2.Konfig.Res_2 := FALSE;
   BB2_AS2.Konfig.Res_3 := FALSE;
   BB2_AS2.Konfig.Res_4 := FALSE;
   BB2_AS2.Konfig.Res_5 := FALSE;
   BB2_AS2.Konfig.Res_6 := FALSE;
   BB2_AS2.Konfig.Res_7 := FALSE;
   BB2_AS2.Konfig.Res_8 := FALSE;
   BB2_AS2.Konfig.Res_9 := FALSE;
   BB2_AS2.Konfig.Res_10 := FALSE;
   BB2_AS2.Konfig.Res_11 := FALSE;
   BB2_AS2.Konfig.Res_12 := FALSE;
   BB2_AS2.Konfig.Res_13 := FALSE;
   BB2_AS2.Konfig.Res_14 := FALSE;
   BB2_AS2.Konfig.Res_15 := FALSE;
   BB2_AS2.Konfig.Res_16 := FALSE;
   BB2_AS2.Konfig.Res_17 := FALSE;
   BB2_AS2.Konfig.Res_18 := FALSE;
   BB2_AS2.Konfig.Res_19 := FALSE;
   BB2_AS2.Konfig.Res_20 := FALSE;
   BB2_AS2.Konfig.Res_21 := FALSE;
   BB2_AS2.Konfig.Res_22 := FALSE;
   BB2_AS2.Konfig.Res_23 := FALSE;
   BB2_AS2.Konfig.Res_24 := FALSE;
   BB2_AS2.Konfig.Res_25 := FALSE;
   BB2_AS2.Konfig.Res_26 := FALSE;
   BB2_AS2.Konfig.Res_27 := FALSE;
   BB2_AS2.Konfig.Res_28 := FALSE;
   BB2_AS2.Konfig.Res_29 := FALSE;
   BB2_AS2.Konfig.Res_30 := FALSE;
   BB2_AS2.Konfig.Prm_Set := FALSE;
   BB2_AS2.P_nenn := 1.0;
   BB2_AS2.EZ_max := 0;
   BB2_AS2.AZ_min := 5;
   BB2_AS2.AZ_Rev := 10;
   BB2_AS2.VZ_St := 5;
   BB2_AS2.UeZ_Endl := 120;
   BB2_AS2.UeZ_BF := 15;
   BB2_AS2.Prio_NS := 0;
   BB2_AS2.Prio_ECS := 0;
   BB2_AS2.Prio_NA := 0;
   BB2_AS2.ESV_NA := 5;
   BB2_SR1.Konfig.Res_0 := FALSE;
   BB2_SR1.Konfig.Res_1 := FALSE;
   BB2_SR1.Konfig.Res_2 := FALSE;
   BB2_SR1.Konfig.Res_3 := FALSE;
   BB2_SR1.Konfig.Res_4 := FALSE;
   BB2_SR1.Konfig.Res_5 := FALSE;
   BB2_SR1.Konfig.Res_6 := FALSE;
   BB2_SR1.Konfig.Res_7 := FALSE;
   BB2_SR1.Konfig.Res_8 := FALSE;
   BB2_SR1.Konfig.Res_9 := FALSE;
   BB2_SR1.Konfig.Res_10 := FALSE;
   BB2_SR1.Konfig.Res_11 := FALSE;
   BB2_SR1.Konfig.Res_12 := FALSE;
   BB2_SR1.Konfig.Res_13 := FALSE;
   BB2_SR1.Konfig.Res_14 := FALSE;
   BB2_SR1.Konfig.Res_15 := FALSE;
   BB2_SR1.Konfig.Res_16 := FALSE;
   BB2_SR1.Konfig.Res_17 := FALSE;
   BB2_SR1.Konfig.Res_18 := FALSE;
   BB2_SR1.Konfig.Res_19 := FALSE;
   BB2_SR1.Konfig.Res_20 := FALSE;
   BB2_SR1.Konfig.Res_21 := FALSE;
   BB2_SR1.Konfig.Res_22 := FALSE;
   BB2_SR1.Konfig.Res_23 := FALSE;
   BB2_SR1.Konfig.Res_24 := FALSE;
   BB2_SR1.Konfig.Res_25 := FALSE;
   BB2_SR1.Konfig.Res_26 := FALSE;
   BB2_SR1.Konfig.Res_27 := FALSE;
   BB2_SR1.Konfig.Res_28 := FALSE;
   BB2_SR1.Konfig.Res_29 := FALSE;
   BB2_SR1.Konfig.Res_30 := FALSE;
   BB2_SR1.Konfig.Prm_Set := FALSE;
   BB2_SR1.P_nenn := 1.0;
   BB2_SR1.EZ_max := 0;
   BB2_SR1.AZ_min := 5;
   BB2_SR1.AZ_Rev := 10;
   BB2_SR1.VZ_St := 5;
   BB2_SR1.UeZ_Endl := 120;
   BB2_SR1.UeZ_BF := 0;
   BB2_SR1.Prio_NS := 0;
   BB2_SR1.Prio_ECS := 0;
   BB2_SR1.Prio_NA := 0;
   BB2_SR1.ESV_NA := 5;
   BB2_SR2.Konfig.Res_0 := FALSE;
   BB2_SR2.Konfig.Res_1 := FALSE;
   BB2_SR2.Konfig.Res_2 := FALSE;
   BB2_SR2.Konfig.Res_3 := FALSE;
   BB2_SR2.Konfig.Res_4 := FALSE;
   BB2_SR2.Konfig.Res_5 := FALSE;
   BB2_SR2.Konfig.Res_6 := FALSE;
   BB2_SR2.Konfig.Res_7 := FALSE;
   BB2_SR2.Konfig.Res_8 := FALSE;
   BB2_SR2.Konfig.Res_9 := FALSE;
   BB2_SR2.Konfig.Res_10 := FALSE;
   BB2_SR2.Konfig.Res_11 := FALSE;
   BB2_SR2.Konfig.Res_12 := FALSE;
   BB2_SR2.Konfig.Res_13 := FALSE;
   BB2_SR2.Konfig.Res_14 := FALSE;
   BB2_SR2.Konfig.Res_15 := FALSE;
   BB2_SR2.Konfig.Res_16 := FALSE;
   BB2_SR2.Konfig.Res_17 := FALSE;
   BB2_SR2.Konfig.Res_18 := FALSE;
   BB2_SR2.Konfig.Res_19 := FALSE;
   BB2_SR2.Konfig.Res_20 := FALSE;
   BB2_SR2.Konfig.Res_21 := FALSE;
   BB2_SR2.Konfig.Res_22 := FALSE;
   BB2_SR2.Konfig.Res_23 := FALSE;
   BB2_SR2.Konfig.Res_24 := FALSE;
   BB2_SR2.Konfig.Res_25 := FALSE;
   BB2_SR2.Konfig.Res_26 := FALSE;
   BB2_SR2.Konfig.Res_27 := FALSE;
   BB2_SR2.Konfig.Res_28 := FALSE;
   BB2_SR2.Konfig.Res_29 := FALSE;
   BB2_SR2.Konfig.Res_30 := FALSE;
   BB2_SR2.Konfig.Prm_Set := FALSE;
   BB2_SR2.P_nenn := 1.0;
   BB2_SR2.EZ_max := 0;
   BB2_SR2.AZ_min := 5;
   BB2_SR2.AZ_Rev := 10;
   BB2_SR2.VZ_St := 5;
   BB2_SR2.UeZ_Endl := 120;
   BB2_SR2.UeZ_BF := 15;
   BB2_SR2.Prio_NS := 0;
   BB2_SR2.Prio_ECS := 0;
   BB2_SR2.Prio_NA := 0;
   BB2_SR2.ESV_NA := 5;
   BB1_SR_K.Konfig.Res_0 := FALSE;
   BB1_SR_K.Konfig.Res_1 := FALSE;
   BB1_SR_K.Konfig.Res_2 := FALSE;
   BB1_SR_K.Konfig.Res_3 := FALSE;
   BB1_SR_K.Konfig.Res_4 := FALSE;
   BB1_SR_K.Konfig.Res_5 := FALSE;
   BB1_SR_K.Konfig.Res_6 := FALSE;
   BB1_SR_K.Konfig.Res_7 := FALSE;
   BB1_SR_K.Konfig.Res_8 := FALSE;
   BB1_SR_K.Konfig.Res_9 := FALSE;
   BB1_SR_K.Konfig.Res_10 := FALSE;
   BB1_SR_K.Konfig.Res_11 := FALSE;
   BB1_SR_K.Konfig.Res_12 := FALSE;
   BB1_SR_K.Konfig.Res_13 := FALSE;
   BB1_SR_K.Konfig.Res_14 := FALSE;
   BB1_SR_K.Konfig.Res_15 := FALSE;
   BB1_SR_K.Konfig.Res_16 := FALSE;
   BB1_SR_K.Konfig.Res_17 := FALSE;
   BB1_SR_K.Konfig.Res_18 := FALSE;
   BB1_SR_K.Konfig.Res_19 := FALSE;
   BB1_SR_K.Konfig.Res_20 := FALSE;
   BB1_SR_K.Konfig.Res_21 := FALSE;
   BB1_SR_K.Konfig.Res_22 := FALSE;
   BB1_SR_K.Konfig.Res_23 := FALSE;
   BB1_SR_K.Konfig.Res_24 := FALSE;
   BB1_SR_K.Konfig.Res_25 := FALSE;
   BB1_SR_K.Konfig.Res_26 := FALSE;
   BB1_SR_K.Konfig.Res_27 := FALSE;
   BB1_SR_K.Konfig.Res_28 := FALSE;
   BB1_SR_K.Konfig.Res_29 := FALSE;
   BB1_SR_K.Konfig.Res_30 := FALSE;
   BB1_SR_K.Konfig.Prm_Set := FALSE;
   BB1_SR_K.P_nenn := 1.0;
   BB1_SR_K.EZ_max := 0;
   BB1_SR_K.AZ_min := 5;
   BB1_SR_K.AZ_Rev := 10;
   BB1_SR_K.VZ_St := 5;
   BB1_SR_K.UeZ_Endl := 120;
   BB1_SR_K.UeZ_BF := 15;
   BB1_SR_K.Prio_NS := 0;
   BB1_SR_K.Prio_ECS := 0;
   BB1_SR_K.Prio_NA := 0;
   BB1_SR_K.ESV_NA := 5;
   Zulauf_AR_P1.Konfig.Res_0 := FALSE;
   Zulauf_AR_P1.Konfig.Res_1 := FALSE;
   Zulauf_AR_P1.Konfig.Res_2 := FALSE;
   Zulauf_AR_P1.Konfig.Res_3 := FALSE;
   Zulauf_AR_P1.Konfig.Res_4 := FALSE;
   Zulauf_AR_P1.Konfig.Res_5 := FALSE;
   Zulauf_AR_P1.Konfig.Res_6 := FALSE;
   Zulauf_AR_P1.Konfig.Res_7 := FALSE;
   Zulauf_AR_P1.Konfig.Res_8 := FALSE;
   Zulauf_AR_P1.Konfig.Res_9 := FALSE;
   Zulauf_AR_P1.Konfig.Res_10 := FALSE;
   Zulauf_AR_P1.Konfig.Res_11 := FALSE;
   Zulauf_AR_P1.Konfig.Res_12 := FALSE;
   Zulauf_AR_P1.Konfig.Res_13 := FALSE;
   Zulauf_AR_P1.Konfig.Res_14 := FALSE;
   Zulauf_AR_P1.Konfig.Res_15 := FALSE;
   Zulauf_AR_P1.Konfig.Res_16 := FALSE;
   Zulauf_AR_P1.Konfig.Res_17 := FALSE;
   Zulauf_AR_P1.Konfig.Res_18 := FALSE;
   Zulauf_AR_P1.Konfig.Res_19 := FALSE;
   Zulauf_AR_P1.Konfig.Res_20 := FALSE;
   Zulauf_AR_P1.Konfig.Res_21 := FALSE;
   Zulauf_AR_P1.Konfig.Res_22 := FALSE;
   Zulauf_AR_P1.Konfig.Res_23 := FALSE;
   Zulauf_AR_P1.Konfig.Res_24 := FALSE;
   Zulauf_AR_P1.Konfig.Res_25 := FALSE;
   Zulauf_AR_P1.Konfig.Res_26 := FALSE;
   Zulauf_AR_P1.Konfig.Res_27 := FALSE;
   Zulauf_AR_P1.Konfig.Res_28 := FALSE;
   Zulauf_AR_P1.Konfig.Res_29 := FALSE;
   Zulauf_AR_P1.Konfig.Res_30 := FALSE;
   Zulauf_AR_P1.Konfig.Prm_Set := FALSE;
   Zulauf_AR_P1.P_nenn := 1.0;
   Zulauf_AR_P1.EZ_max := 0;
   Zulauf_AR_P1.AZ_min := 5;
   Zulauf_AR_P1.AZ_Rev := 10;
   Zulauf_AR_P1.VZ_St := 5;
   Zulauf_AR_P1.UeZ_Endl := 120;
   Zulauf_AR_P1.UeZ_BF := 15;
   Zulauf_AR_P1.Prio_NS := 0;
   Zulauf_AR_P1.Prio_ECS := 0;
   Zulauf_AR_P1.Prio_NA := 0;
   Zulauf_AR_P1.ESV_NA := 5;
   Zulauf_AR_P2.Konfig.Res_0 := FALSE;
   Zulauf_AR_P2.Konfig.Res_1 := FALSE;
   Zulauf_AR_P2.Konfig.Res_2 := FALSE;
   Zulauf_AR_P2.Konfig.Res_3 := FALSE;
   Zulauf_AR_P2.Konfig.Res_4 := FALSE;
   Zulauf_AR_P2.Konfig.Res_5 := FALSE;
   Zulauf_AR_P2.Konfig.Res_6 := FALSE;
   Zulauf_AR_P2.Konfig.Res_7 := FALSE;
   Zulauf_AR_P2.Konfig.Res_8 := FALSE;
   Zulauf_AR_P2.Konfig.Res_9 := FALSE;
   Zulauf_AR_P2.Konfig.Res_10 := FALSE;
   Zulauf_AR_P2.Konfig.Res_11 := FALSE;
   Zulauf_AR_P2.Konfig.Res_12 := FALSE;
   Zulauf_AR_P2.Konfig.Res_13 := FALSE;
   Zulauf_AR_P2.Konfig.Res_14 := FALSE;
   Zulauf_AR_P2.Konfig.Res_15 := FALSE;
   Zulauf_AR_P2.Konfig.Res_16 := FALSE;
   Zulauf_AR_P2.Konfig.Res_17 := FALSE;
   Zulauf_AR_P2.Konfig.Res_18 := FALSE;
   Zulauf_AR_P2.Konfig.Res_19 := FALSE;
   Zulauf_AR_P2.Konfig.Res_20 := FALSE;
   Zulauf_AR_P2.Konfig.Res_21 := FALSE;
   Zulauf_AR_P2.Konfig.Res_22 := FALSE;
   Zulauf_AR_P2.Konfig.Res_23 := FALSE;
   Zulauf_AR_P2.Konfig.Res_24 := FALSE;
   Zulauf_AR_P2.Konfig.Res_25 := FALSE;
   Zulauf_AR_P2.Konfig.Res_26 := FALSE;
   Zulauf_AR_P2.Konfig.Res_27 := FALSE;
   Zulauf_AR_P2.Konfig.Res_28 := FALSE;
   Zulauf_AR_P2.Konfig.Res_29 := FALSE;
   Zulauf_AR_P2.Konfig.Res_30 := FALSE;
   Zulauf_AR_P2.Konfig.Prm_Set := FALSE;
   Zulauf_AR_P2.P_nenn := 1.0;
   Zulauf_AR_P2.EZ_max := 0;
   Zulauf_AR_P2.AZ_min := 5;
   Zulauf_AR_P2.AZ_Rev := 10;
   Zulauf_AR_P2.VZ_St := 5;
   Zulauf_AR_P2.UeZ_Endl := 120;
   Zulauf_AR_P2.UeZ_BF := 15;
   Zulauf_AR_P2.Prio_NS := 0;
   Zulauf_AR_P2.Prio_ECS := 0;
   Zulauf_AR_P2.Prio_NA := 0;
   Zulauf_AR_P2.ESV_NA := 5;
   Zulauf_AS.Konfig.Res_0 := FALSE;
   Zulauf_AS.Konfig.Res_1 := FALSE;
   Zulauf_AS.Konfig.Res_2 := FALSE;
   Zulauf_AS.Konfig.Res_3 := FALSE;
   Zulauf_AS.Konfig.Res_4 := FALSE;
   Zulauf_AS.Konfig.Res_5 := FALSE;
   Zulauf_AS.Konfig.Res_6 := FALSE;
   Zulauf_AS.Konfig.Res_7 := FALSE;
   Zulauf_AS.Konfig.Res_8 := FALSE;
   Zulauf_AS.Konfig.Res_9 := FALSE;
   Zulauf_AS.Konfig.Res_10 := FALSE;
   Zulauf_AS.Konfig.Res_11 := FALSE;
   Zulauf_AS.Konfig.Res_12 := FALSE;
   Zulauf_AS.Konfig.Res_13 := FALSE;
   Zulauf_AS.Konfig.Res_14 := FALSE;
   Zulauf_AS.Konfig.Res_15 := FALSE;
   Zulauf_AS.Konfig.Res_16 := FALSE;
   Zulauf_AS.Konfig.Res_17 := FALSE;
   Zulauf_AS.Konfig.Res_18 := FALSE;
   Zulauf_AS.Konfig.Res_19 := FALSE;
   Zulauf_AS.Konfig.Res_20 := FALSE;
   Zulauf_AS.Konfig.Res_21 := FALSE;
   Zulauf_AS.Konfig.Res_22 := FALSE;
   Zulauf_AS.Konfig.Res_23 := FALSE;
   Zulauf_AS.Konfig.Res_24 := FALSE;
   Zulauf_AS.Konfig.Res_25 := FALSE;
   Zulauf_AS.Konfig.Res_26 := FALSE;
   Zulauf_AS.Konfig.Res_27 := FALSE;
   Zulauf_AS.Konfig.Res_28 := FALSE;
   Zulauf_AS.Konfig.Res_29 := FALSE;
   Zulauf_AS.Konfig.Res_30 := FALSE;
   Zulauf_AS.Konfig.Prm_Set := FALSE;
   Zulauf_AS.P_nenn := 1.0;
   Zulauf_AS.EZ_max := 0;
   Zulauf_AS.AZ_min := 5;
   Zulauf_AS.AZ_Rev := 10;
   Zulauf_AS.VZ_St := 5;
   Zulauf_AS.UeZ_Endl := 120;
   Zulauf_AS.UeZ_BF := 15;
   Zulauf_AS.Prio_NS := 0;
   Zulauf_AS.Prio_ECS := 0;
   Zulauf_AS.Prio_NA := 0;
   Zulauf_AS.ESV_NA := 5;
   Zulauf_RA_SA.Konfig.Res_0 := FALSE;
   Zulauf_RA_SA.Konfig.Res_1 := FALSE;
   Zulauf_RA_SA.Konfig.Res_2 := FALSE;
   Zulauf_RA_SA.Konfig.Res_3 := FALSE;
   Zulauf_RA_SA.Konfig.Res_4 := FALSE;
   Zulauf_RA_SA.Konfig.Res_5 := FALSE;
   Zulauf_RA_SA.Konfig.Res_6 := FALSE;
   Zulauf_RA_SA.Konfig.Res_7 := FALSE;
   Zulauf_RA_SA.Konfig.Res_8 := FALSE;
   Zulauf_RA_SA.Konfig.Res_9 := FALSE;
   Zulauf_RA_SA.Konfig.Res_10 := FALSE;
   Zulauf_RA_SA.Konfig.Res_11 := FALSE;
   Zulauf_RA_SA.Konfig.Res_12 := FALSE;
   Zulauf_RA_SA.Konfig.Res_13 := FALSE;
   Zulauf_RA_SA.Konfig.Res_14 := FALSE;
   Zulauf_RA_SA.Konfig.Res_15 := FALSE;
   Zulauf_RA_SA.Konfig.Res_16 := FALSE;
   Zulauf_RA_SA.Konfig.Res_17 := FALSE;
   Zulauf_RA_SA.Konfig.Res_18 := FALSE;
   Zulauf_RA_SA.Konfig.Res_19 := FALSE;
   Zulauf_RA_SA.Konfig.Res_20 := FALSE;
   Zulauf_RA_SA.Konfig.Res_21 := FALSE;
   Zulauf_RA_SA.Konfig.Res_22 := FALSE;
   Zulauf_RA_SA.Konfig.Res_23 := FALSE;
   Zulauf_RA_SA.Konfig.Res_24 := FALSE;
   Zulauf_RA_SA.Konfig.Res_25 := FALSE;
   Zulauf_RA_SA.Konfig.Res_26 := FALSE;
   Zulauf_RA_SA.Konfig.Res_27 := FALSE;
   Zulauf_RA_SA.Konfig.Res_28 := FALSE;
   Zulauf_RA_SA.Konfig.Res_29 := FALSE;
   Zulauf_RA_SA.Konfig.Res_30 := FALSE;
   Zulauf_RA_SA.Konfig.Prm_Set := FALSE;
   Zulauf_RA_SA.P_nenn := 1.0;
   Zulauf_RA_SA.EZ_max := 0;
   Zulauf_RA_SA.AZ_min := 5;
   Zulauf_RA_SA.AZ_Rev := 10;
   Zulauf_RA_SA.VZ_St := 5;
   Zulauf_RA_SA.UeZ_Endl := 120;
   Zulauf_RA_SA.UeZ_BF := 15;
   Zulauf_RA_SA.Prio_NS := 0;
   Zulauf_RA_SA.Prio_ECS := 0;
   Zulauf_RA_SA.Prio_NA := 0;
   Zulauf_RA_SA.ESV_NA := 5;
   Zulauf_RA_HZS.Konfig.Res_0 := FALSE;
   Zulauf_RA_HZS.Konfig.Res_1 := FALSE;
   Zulauf_RA_HZS.Konfig.Res_2 := FALSE;
   Zulauf_RA_HZS.Konfig.Res_3 := FALSE;
   Zulauf_RA_HZS.Konfig.Res_4 := FALSE;
   Zulauf_RA_HZS.Konfig.Res_5 := FALSE;
   Zulauf_RA_HZS.Konfig.Res_6 := FALSE;
   Zulauf_RA_HZS.Konfig.Res_7 := FALSE;
   Zulauf_RA_HZS.Konfig.Res_8 := FALSE;
   Zulauf_RA_HZS.Konfig.Res_9 := FALSE;
   Zulauf_RA_HZS.Konfig.Res_10 := FALSE;
   Zulauf_RA_HZS.Konfig.Res_11 := FALSE;
   Zulauf_RA_HZS.Konfig.Res_12 := FALSE;
   Zulauf_RA_HZS.Konfig.Res_13 := FALSE;
   Zulauf_RA_HZS.Konfig.Res_14 := FALSE;
   Zulauf_RA_HZS.Konfig.Res_15 := FALSE;
   Zulauf_RA_HZS.Konfig.Res_16 := FALSE;
   Zulauf_RA_HZS.Konfig.Res_17 := FALSE;
   Zulauf_RA_HZS.Konfig.Res_18 := FALSE;
   Zulauf_RA_HZS.Konfig.Res_19 := FALSE;
   Zulauf_RA_HZS.Konfig.Res_20 := FALSE;
   Zulauf_RA_HZS.Konfig.Res_21 := FALSE;
   Zulauf_RA_HZS.Konfig.Res_22 := FALSE;
   Zulauf_RA_HZS.Konfig.Res_23 := FALSE;
   Zulauf_RA_HZS.Konfig.Res_24 := FALSE;
   Zulauf_RA_HZS.Konfig.Res_25 := FALSE;
   Zulauf_RA_HZS.Konfig.Res_26 := FALSE;
   Zulauf_RA_HZS.Konfig.Res_27 := FALSE;
   Zulauf_RA_HZS.Konfig.Res_28 := FALSE;
   Zulauf_RA_HZS.Konfig.Res_29 := FALSE;
   Zulauf_RA_HZS.Konfig.Res_30 := FALSE;
   Zulauf_RA_HZS.Konfig.Prm_Set := FALSE;
   Zulauf_RA_HZS.P_nenn := 1.0;
   Zulauf_RA_HZS.EZ_max := 0;
   Zulauf_RA_HZS.AZ_min := 5;
   Zulauf_RA_HZS.AZ_Rev := 10;
   Zulauf_RA_HZS.VZ_St := 5;
   Zulauf_RA_HZS.UeZ_Endl := 120;
   Zulauf_RA_HZS.UeZ_BF := 15;
   Zulauf_RA_HZS.Prio_NS := 0;
   Zulauf_RA_HZS.Prio_ECS := 0;
   Zulauf_RA_HZS.Prio_NA := 0;
   Zulauf_RA_HZS.ESV_NA := 5;
   Zulauf_RA_VKS.Konfig.Res_0 := FALSE;
   Zulauf_RA_VKS.Konfig.Res_1 := FALSE;
   Zulauf_RA_VKS.Konfig.Res_2 := FALSE;
   Zulauf_RA_VKS.Konfig.Res_3 := FALSE;
   Zulauf_RA_VKS.Konfig.Res_4 := FALSE;
   Zulauf_RA_VKS.Konfig.Res_5 := FALSE;
   Zulauf_RA_VKS.Konfig.Res_6 := FALSE;
   Zulauf_RA_VKS.Konfig.Res_7 := FALSE;
   Zulauf_RA_VKS.Konfig.Res_8 := FALSE;
   Zulauf_RA_VKS.Konfig.Res_9 := FALSE;
   Zulauf_RA_VKS.Konfig.Res_10 := FALSE;
   Zulauf_RA_VKS.Konfig.Res_11 := FALSE;
   Zulauf_RA_VKS.Konfig.Res_12 := FALSE;
   Zulauf_RA_VKS.Konfig.Res_13 := FALSE;
   Zulauf_RA_VKS.Konfig.Res_14 := FALSE;
   Zulauf_RA_VKS.Konfig.Res_15 := FALSE;
   Zulauf_RA_VKS.Konfig.Res_16 := FALSE;
   Zulauf_RA_VKS.Konfig.Res_17 := FALSE;
   Zulauf_RA_VKS.Konfig.Res_18 := FALSE;
   Zulauf_RA_VKS.Konfig.Res_19 := FALSE;
   Zulauf_RA_VKS.Konfig.Res_20 := FALSE;
   Zulauf_RA_VKS.Konfig.Res_21 := FALSE;
   Zulauf_RA_VKS.Konfig.Res_22 := FALSE;
   Zulauf_RA_VKS.Konfig.Res_23 := FALSE;
   Zulauf_RA_VKS.Konfig.Res_24 := FALSE;
   Zulauf_RA_VKS.Konfig.Res_25 := FALSE;
   Zulauf_RA_VKS.Konfig.Res_26 := FALSE;
   Zulauf_RA_VKS.Konfig.Res_27 := FALSE;
   Zulauf_RA_VKS.Konfig.Res_28 := FALSE;
   Zulauf_RA_VKS.Konfig.Res_29 := FALSE;
   Zulauf_RA_VKS.Konfig.Res_30 := FALSE;
   Zulauf_RA_VKS.Konfig.Prm_Set := FALSE;
   Zulauf_RA_VKS.P_nenn := 1.0;
   Zulauf_RA_VKS.EZ_max := 0;
   Zulauf_RA_VKS.AZ_min := 5;
   Zulauf_RA_VKS.AZ_Rev := 10;
   Zulauf_RA_VKS.VZ_St := 5;
   Zulauf_RA_VKS.UeZ_Endl := 120;
   Zulauf_RA_VKS.UeZ_BF := 15;
   Zulauf_RA_VKS.Prio_NS := 0;
   Zulauf_RA_VKS.Prio_ECS := 0;
   Zulauf_RA_VKS.Prio_NA := 0;
   Zulauf_RA_VKS.ESV_NA := 5;
   Zulauf_RA_V.Konfig.Res_0 := FALSE;
   Zulauf_RA_V.Konfig.Res_1 := FALSE;
   Zulauf_RA_V.Konfig.Res_2 := FALSE;
   Zulauf_RA_V.Konfig.Res_3 := FALSE;
   Zulauf_RA_V.Konfig.Res_4 := FALSE;
   Zulauf_RA_V.Konfig.Res_5 := FALSE;
   Zulauf_RA_V.Konfig.Res_6 := FALSE;
   Zulauf_RA_V.Konfig.Res_7 := FALSE;
   Zulauf_RA_V.Konfig.Res_8 := FALSE;
   Zulauf_RA_V.Konfig.Res_9 := FALSE;
   Zulauf_RA_V.Konfig.Res_10 := FALSE;
   Zulauf_RA_V.Konfig.Res_11 := FALSE;
   Zulauf_RA_V.Konfig.Res_12 := FALSE;
   Zulauf_RA_V.Konfig.Res_13 := FALSE;
   Zulauf_RA_V.Konfig.Res_14 := FALSE;
   Zulauf_RA_V.Konfig.Res_15 := FALSE;
   Zulauf_RA_V.Konfig.Res_16 := FALSE;
   Zulauf_RA_V.Konfig.Res_17 := FALSE;
   Zulauf_RA_V.Konfig.Res_18 := FALSE;
   Zulauf_RA_V.Konfig.Res_19 := FALSE;
   Zulauf_RA_V.Konfig.Res_20 := FALSE;
   Zulauf_RA_V.Konfig.Res_21 := FALSE;
   Zulauf_RA_V.Konfig.Res_22 := FALSE;
   Zulauf_RA_V.Konfig.Res_23 := FALSE;
   Zulauf_RA_V.Konfig.Res_24 := FALSE;
   Zulauf_RA_V.Konfig.Res_25 := FALSE;
   Zulauf_RA_V.Konfig.Res_26 := FALSE;
   Zulauf_RA_V.Konfig.Res_27 := FALSE;
   Zulauf_RA_V.Konfig.Res_28 := FALSE;
   Zulauf_RA_V.Konfig.Res_29 := FALSE;
   Zulauf_RA_V.Konfig.Res_30 := FALSE;
   Zulauf_RA_V.Konfig.Prm_Set := FALSE;
   Zulauf_RA_V.P_nenn := 1.0;
   Zulauf_RA_V.EZ_max := 0;
   Zulauf_RA_V.AZ_min := 5;
   Zulauf_RA_V.AZ_Rev := 10;
   Zulauf_RA_V.VZ_St := 5;
   Zulauf_RA_V.UeZ_Endl := 120;
   Zulauf_RA_V.UeZ_BF := 15;
   Zulauf_RA_V.Prio_NS := 0;
   Zulauf_RA_V.Prio_ECS := 0;
   Zulauf_RA_V.Prio_NA := 0;
   Zulauf_RA_V.ESV_NA := 5;
   Zulauf_RA_RP.Konfig.Res_0 := FALSE;
   Zulauf_RA_RP.Konfig.Res_1 := FALSE;
   Zulauf_RA_RP.Konfig.Res_2 := FALSE;
   Zulauf_RA_RP.Konfig.Res_3 := FALSE;
   Zulauf_RA_RP.Konfig.Res_4 := FALSE;
   Zulauf_RA_RP.Konfig.Res_5 := FALSE;
   Zulauf_RA_RP.Konfig.Res_6 := FALSE;
   Zulauf_RA_RP.Konfig.Res_7 := FALSE;
   Zulauf_RA_RP.Konfig.Res_8 := FALSE;
   Zulauf_RA_RP.Konfig.Res_9 := FALSE;
   Zulauf_RA_RP.Konfig.Res_10 := FALSE;
   Zulauf_RA_RP.Konfig.Res_11 := FALSE;
   Zulauf_RA_RP.Konfig.Res_12 := FALSE;
   Zulauf_RA_RP.Konfig.Res_13 := FALSE;
   Zulauf_RA_RP.Konfig.Res_14 := FALSE;
   Zulauf_RA_RP.Konfig.Res_15 := FALSE;
   Zulauf_RA_RP.Konfig.Res_16 := FALSE;
   Zulauf_RA_RP.Konfig.Res_17 := FALSE;
   Zulauf_RA_RP.Konfig.Res_18 := FALSE;
   Zulauf_RA_RP.Konfig.Res_19 := FALSE;
   Zulauf_RA_RP.Konfig.Res_20 := FALSE;
   Zulauf_RA_RP.Konfig.Res_21 := FALSE;
   Zulauf_RA_RP.Konfig.Res_22 := FALSE;
   Zulauf_RA_RP.Konfig.Res_23 := FALSE;
   Zulauf_RA_RP.Konfig.Res_24 := FALSE;
   Zulauf_RA_RP.Konfig.Res_25 := FALSE;
   Zulauf_RA_RP.Konfig.Res_26 := FALSE;
   Zulauf_RA_RP.Konfig.Res_27 := FALSE;
   Zulauf_RA_RP.Konfig.Res_28 := FALSE;
   Zulauf_RA_RP.Konfig.Res_29 := FALSE;
   Zulauf_RA_RP.Konfig.Res_30 := FALSE;
   Zulauf_RA_RP.Konfig.Prm_Set := FALSE;
   Zulauf_RA_RP.P_nenn := 1.0;
   Zulauf_RA_RP.EZ_max := 0;
   Zulauf_RA_RP.AZ_min := 5;
   Zulauf_RA_RP.AZ_Rev := 10;
   Zulauf_RA_RP.VZ_St := 5;
   Zulauf_RA_RP.UeZ_Endl := 120;
   Zulauf_RA_RP.UeZ_BF := 15;
   Zulauf_RA_RP.Prio_NS := 0;
   Zulauf_RA_RP.Prio_ECS := 0;
   Zulauf_RA_RP.Prio_NA := 0;
   Zulauf_RA_RP.ESV_NA := 5;
   Zulauf_RA_FP.Konfig.Res_0 := FALSE;
   Zulauf_RA_FP.Konfig.Res_1 := FALSE;
   Zulauf_RA_FP.Konfig.Res_2 := FALSE;
   Zulauf_RA_FP.Konfig.Res_3 := FALSE;
   Zulauf_RA_FP.Konfig.Res_4 := FALSE;
   Zulauf_RA_FP.Konfig.Res_5 := FALSE;
   Zulauf_RA_FP.Konfig.Res_6 := FALSE;
   Zulauf_RA_FP.Konfig.Res_7 := FALSE;
   Zulauf_RA_FP.Konfig.Res_8 := FALSE;
   Zulauf_RA_FP.Konfig.Res_9 := FALSE;
   Zulauf_RA_FP.Konfig.Res_10 := FALSE;
   Zulauf_RA_FP.Konfig.Res_11 := FALSE;
   Zulauf_RA_FP.Konfig.Res_12 := FALSE;
   Zulauf_RA_FP.Konfig.Res_13 := FALSE;
   Zulauf_RA_FP.Konfig.Res_14 := FALSE;
   Zulauf_RA_FP.Konfig.Res_15 := FALSE;
   Zulauf_RA_FP.Konfig.Res_16 := FALSE;
   Zulauf_RA_FP.Konfig.Res_17 := FALSE;
   Zulauf_RA_FP.Konfig.Res_18 := FALSE;
   Zulauf_RA_FP.Konfig.Res_19 := FALSE;
   Zulauf_RA_FP.Konfig.Res_20 := FALSE;
   Zulauf_RA_FP.Konfig.Res_21 := FALSE;
   Zulauf_RA_FP.Konfig.Res_22 := FALSE;
   Zulauf_RA_FP.Konfig.Res_23 := FALSE;
   Zulauf_RA_FP.Konfig.Res_24 := FALSE;
   Zulauf_RA_FP.Konfig.Res_25 := FALSE;
   Zulauf_RA_FP.Konfig.Res_26 := FALSE;
   Zulauf_RA_FP.Konfig.Res_27 := FALSE;
   Zulauf_RA_FP.Konfig.Res_28 := FALSE;
   Zulauf_RA_FP.Konfig.Res_29 := FALSE;
   Zulauf_RA_FP.Konfig.Res_30 := FALSE;
   Zulauf_RA_FP.Konfig.Prm_Set := FALSE;
   Zulauf_RA_FP.P_nenn := 1.0;
   Zulauf_RA_FP.EZ_max := 0;
   Zulauf_RA_FP.AZ_min := 5;
   Zulauf_RA_FP.AZ_Rev := 10;
   Zulauf_RA_FP.VZ_St := 5;
   Zulauf_RA_FP.UeZ_Endl := 120;
   Zulauf_RA_FP.UeZ_BF := 15;
   Zulauf_RA_FP.Prio_NS := 0;
   Zulauf_RA_FP.Prio_ECS := 0;
   Zulauf_RA_FP.Prio_NA := 0;
   Zulauf_RA_FP.ESV_NA := 5;
   Schlamm_BP.Konfig.Res_0 := FALSE;
   Schlamm_BP.Konfig.Res_1 := FALSE;
   Schlamm_BP.Konfig.Res_2 := FALSE;
   Schlamm_BP.Konfig.Res_3 := FALSE;
   Schlamm_BP.Konfig.Res_4 := FALSE;
   Schlamm_BP.Konfig.Res_5 := FALSE;
   Schlamm_BP.Konfig.Res_6 := FALSE;
   Schlamm_BP.Konfig.Res_7 := FALSE;
   Schlamm_BP.Konfig.Res_8 := FALSE;
   Schlamm_BP.Konfig.Res_9 := FALSE;
   Schlamm_BP.Konfig.Res_10 := FALSE;
   Schlamm_BP.Konfig.Res_11 := FALSE;
   Schlamm_BP.Konfig.Res_12 := FALSE;
   Schlamm_BP.Konfig.Res_13 := FALSE;
   Schlamm_BP.Konfig.Res_14 := FALSE;
   Schlamm_BP.Konfig.Res_15 := FALSE;
   Schlamm_BP.Konfig.Res_16 := FALSE;
   Schlamm_BP.Konfig.Res_17 := FALSE;
   Schlamm_BP.Konfig.Res_18 := FALSE;
   Schlamm_BP.Konfig.Res_19 := FALSE;
   Schlamm_BP.Konfig.Res_20 := FALSE;
   Schlamm_BP.Konfig.Res_21 := FALSE;
   Schlamm_BP.Konfig.Res_22 := FALSE;
   Schlamm_BP.Konfig.Res_23 := FALSE;
   Schlamm_BP.Konfig.Res_24 := FALSE;
   Schlamm_BP.Konfig.Res_25 := FALSE;
   Schlamm_BP.Konfig.Res_26 := FALSE;
   Schlamm_BP.Konfig.Res_27 := FALSE;
   Schlamm_BP.Konfig.Res_28 := FALSE;
   Schlamm_BP.Konfig.Res_29 := FALSE;
   Schlamm_BP.Konfig.Res_30 := FALSE;
   Schlamm_BP.Konfig.Prm_Set := FALSE;
   Schlamm_BP.P_nenn := 1.0;
   Schlamm_BP.EZ_max := 0;
   Schlamm_BP.AZ_min := 5;
   Schlamm_BP.AZ_Rev := 10;
   Schlamm_BP.VZ_St := 5;
   Schlamm_BP.UeZ_Endl := 120;
   Schlamm_BP.UeZ_BF := 15;
   Schlamm_BP.Prio_NS := 0;
   Schlamm_BP.Prio_ECS := 0;
   Schlamm_BP.Prio_NA := 0;
   Schlamm_BP.ESV_NA := 5;
   Truebwasser_P1.Konfig.Res_0 := FALSE;
   Truebwasser_P1.Konfig.Res_1 := FALSE;
   Truebwasser_P1.Konfig.Res_2 := FALSE;
   Truebwasser_P1.Konfig.Res_3 := FALSE;
   Truebwasser_P1.Konfig.Res_4 := FALSE;
   Truebwasser_P1.Konfig.Res_5 := FALSE;
   Truebwasser_P1.Konfig.Res_6 := FALSE;
   Truebwasser_P1.Konfig.Res_7 := FALSE;
   Truebwasser_P1.Konfig.Res_8 := FALSE;
   Truebwasser_P1.Konfig.Res_9 := FALSE;
   Truebwasser_P1.Konfig.Res_10 := FALSE;
   Truebwasser_P1.Konfig.Res_11 := FALSE;
   Truebwasser_P1.Konfig.Res_12 := FALSE;
   Truebwasser_P1.Konfig.Res_13 := FALSE;
   Truebwasser_P1.Konfig.Res_14 := FALSE;
   Truebwasser_P1.Konfig.Res_15 := FALSE;
   Truebwasser_P1.Konfig.Res_16 := FALSE;
   Truebwasser_P1.Konfig.Res_17 := FALSE;
   Truebwasser_P1.Konfig.Res_18 := FALSE;
   Truebwasser_P1.Konfig.Res_19 := FALSE;
   Truebwasser_P1.Konfig.Res_20 := FALSE;
   Truebwasser_P1.Konfig.Res_21 := FALSE;
   Truebwasser_P1.Konfig.Res_22 := FALSE;
   Truebwasser_P1.Konfig.Res_23 := FALSE;
   Truebwasser_P1.Konfig.Res_24 := FALSE;
   Truebwasser_P1.Konfig.Res_25 := FALSE;
   Truebwasser_P1.Konfig.Res_26 := FALSE;
   Truebwasser_P1.Konfig.Res_27 := FALSE;
   Truebwasser_P1.Konfig.Res_28 := FALSE;
   Truebwasser_P1.Konfig.Res_29 := FALSE;
   Truebwasser_P1.Konfig.Res_30 := FALSE;
   Truebwasser_P1.Konfig.Prm_Set := FALSE;
   Truebwasser_P1.P_nenn := 1.0;
   Truebwasser_P1.EZ_max := 0;
   Truebwasser_P1.AZ_min := 5;
   Truebwasser_P1.AZ_Rev := 10;
   Truebwasser_P1.VZ_St := 5;
   Truebwasser_P1.UeZ_Endl := 120;
   Truebwasser_P1.UeZ_BF := 15;
   Truebwasser_P1.Prio_NS := 0;
   Truebwasser_P1.Prio_ECS := 0;
   Truebwasser_P1.Prio_NA := 0;
   Truebwasser_P1.ESV_NA := 5;
   Truebwasser_P2.Konfig.Res_0 := FALSE;
   Truebwasser_P2.Konfig.Res_1 := FALSE;
   Truebwasser_P2.Konfig.Res_2 := FALSE;
   Truebwasser_P2.Konfig.Res_3 := FALSE;
   Truebwasser_P2.Konfig.Res_4 := FALSE;
   Truebwasser_P2.Konfig.Res_5 := FALSE;
   Truebwasser_P2.Konfig.Res_6 := FALSE;
   Truebwasser_P2.Konfig.Res_7 := FALSE;
   Truebwasser_P2.Konfig.Res_8 := FALSE;
   Truebwasser_P2.Konfig.Res_9 := FALSE;
   Truebwasser_P2.Konfig.Res_10 := FALSE;
   Truebwasser_P2.Konfig.Res_11 := FALSE;
   Truebwasser_P2.Konfig.Res_12 := FALSE;
   Truebwasser_P2.Konfig.Res_13 := FALSE;
   Truebwasser_P2.Konfig.Res_14 := FALSE;
   Truebwasser_P2.Konfig.Res_15 := FALSE;
   Truebwasser_P2.Konfig.Res_16 := FALSE;
   Truebwasser_P2.Konfig.Res_17 := FALSE;
   Truebwasser_P2.Konfig.Res_18 := FALSE;
   Truebwasser_P2.Konfig.Res_19 := FALSE;
   Truebwasser_P2.Konfig.Res_20 := FALSE;
   Truebwasser_P2.Konfig.Res_21 := FALSE;
   Truebwasser_P2.Konfig.Res_22 := FALSE;
   Truebwasser_P2.Konfig.Res_23 := FALSE;
   Truebwasser_P2.Konfig.Res_24 := FALSE;
   Truebwasser_P2.Konfig.Res_25 := FALSE;
   Truebwasser_P2.Konfig.Res_26 := FALSE;
   Truebwasser_P2.Konfig.Res_27 := FALSE;
   Truebwasser_P2.Konfig.Res_28 := FALSE;
   Truebwasser_P2.Konfig.Res_29 := FALSE;
   Truebwasser_P2.Konfig.Res_30 := FALSE;
   Truebwasser_P2.Konfig.Prm_Set := FALSE;
   Truebwasser_P2.P_nenn := 1.0;
   Truebwasser_P2.EZ_max := 0;
   Truebwasser_P2.AZ_min := 5;
   Truebwasser_P2.AZ_Rev := 10;
   Truebwasser_P2.VZ_St := 5;
   Truebwasser_P2.UeZ_Endl := 120;
   Truebwasser_P2.UeZ_BF := 15;
   Truebwasser_P2.Prio_NS := 0;
   Truebwasser_P2.Prio_ECS := 0;
   Truebwasser_P2.Prio_NA := 0;
   Truebwasser_P2.ESV_NA := 5;
   Schlamm_AS.Konfig.Res_0 := FALSE;
   Schlamm_AS.Konfig.Res_1 := FALSE;
   Schlamm_AS.Konfig.Res_2 := FALSE;
   Schlamm_AS.Konfig.Res_3 := FALSE;
   Schlamm_AS.Konfig.Res_4 := FALSE;
   Schlamm_AS.Konfig.Res_5 := FALSE;
   Schlamm_AS.Konfig.Res_6 := FALSE;
   Schlamm_AS.Konfig.Res_7 := FALSE;
   Schlamm_AS.Konfig.Res_8 := FALSE;
   Schlamm_AS.Konfig.Res_9 := FALSE;
   Schlamm_AS.Konfig.Res_10 := FALSE;
   Schlamm_AS.Konfig.Res_11 := FALSE;
   Schlamm_AS.Konfig.Res_12 := FALSE;
   Schlamm_AS.Konfig.Res_13 := FALSE;
   Schlamm_AS.Konfig.Res_14 := FALSE;
   Schlamm_AS.Konfig.Res_15 := FALSE;
   Schlamm_AS.Konfig.Res_16 := FALSE;
   Schlamm_AS.Konfig.Res_17 := FALSE;
   Schlamm_AS.Konfig.Res_18 := FALSE;
   Schlamm_AS.Konfig.Res_19 := FALSE;
   Schlamm_AS.Konfig.Res_20 := FALSE;
   Schlamm_AS.Konfig.Res_21 := FALSE;
   Schlamm_AS.Konfig.Res_22 := FALSE;
   Schlamm_AS.Konfig.Res_23 := FALSE;
   Schlamm_AS.Konfig.Res_24 := FALSE;
   Schlamm_AS.Konfig.Res_25 := FALSE;
   Schlamm_AS.Konfig.Res_26 := FALSE;
   Schlamm_AS.Konfig.Res_27 := FALSE;
   Schlamm_AS.Konfig.Res_28 := FALSE;
   Schlamm_AS.Konfig.Res_29 := FALSE;
   Schlamm_AS.Konfig.Res_30 := FALSE;
   Schlamm_AS.Konfig.Prm_Set := FALSE;
   Schlamm_AS.P_nenn := 1.0;
   Schlamm_AS.EZ_max := 0;
   Schlamm_AS.AZ_min := 5;
   Schlamm_AS.AZ_Rev := 10;
   Schlamm_AS.VZ_St := 5;
   Schlamm_AS.UeZ_Endl := 120;
   Schlamm_AS.UeZ_BF := 15;
   Schlamm_AS.Prio_NS := 0;
   Schlamm_AS.Prio_ECS := 0;
   Schlamm_AS.Prio_NA := 0;
   Schlamm_AS.ESV_NA := 5;
   BB2_SR_K.Konfig.Res_0 := FALSE;
   BB2_SR_K.Konfig.Res_1 := FALSE;
   BB2_SR_K.Konfig.Res_2 := FALSE;
   BB2_SR_K.Konfig.Res_3 := FALSE;
   BB2_SR_K.Konfig.Res_4 := FALSE;
   BB2_SR_K.Konfig.Res_5 := FALSE;
   BB2_SR_K.Konfig.Res_6 := FALSE;
   BB2_SR_K.Konfig.Res_7 := FALSE;
   BB2_SR_K.Konfig.Res_8 := FALSE;
   BB2_SR_K.Konfig.Res_9 := FALSE;
   BB2_SR_K.Konfig.Res_10 := FALSE;
   BB2_SR_K.Konfig.Res_11 := FALSE;
   BB2_SR_K.Konfig.Res_12 := FALSE;
   BB2_SR_K.Konfig.Res_13 := FALSE;
   BB2_SR_K.Konfig.Res_14 := FALSE;
   BB2_SR_K.Konfig.Res_15 := FALSE;
   BB2_SR_K.Konfig.Res_16 := FALSE;
   BB2_SR_K.Konfig.Res_17 := FALSE;
   BB2_SR_K.Konfig.Res_18 := FALSE;
   BB2_SR_K.Konfig.Res_19 := FALSE;
   BB2_SR_K.Konfig.Res_20 := FALSE;
   BB2_SR_K.Konfig.Res_21 := FALSE;
   BB2_SR_K.Konfig.Res_22 := FALSE;
   BB2_SR_K.Konfig.Res_23 := FALSE;
   BB2_SR_K.Konfig.Res_24 := FALSE;
   BB2_SR_K.Konfig.Res_25 := FALSE;
   BB2_SR_K.Konfig.Res_26 := FALSE;
   BB2_SR_K.Konfig.Res_27 := FALSE;
   BB2_SR_K.Konfig.Res_28 := FALSE;
   BB2_SR_K.Konfig.Res_29 := FALSE;
   BB2_SR_K.Konfig.Res_30 := FALSE;
   BB2_SR_K.Konfig.Prm_Set := FALSE;
   BB2_SR_K.P_nenn := 1.0;
   BB2_SR_K.EZ_max := 0;
   BB2_SR_K.AZ_min := 5;
   BB2_SR_K.AZ_Rev := 10;
   BB2_SR_K.VZ_St := 5;
   BB2_SR_K.UeZ_Endl := 120;
   BB2_SR_K.UeZ_BF := 15;
   BB2_SR_K.Prio_NS := 0;
   BB2_SR_K.Prio_ECS := 0;
   BB2_SR_K.Prio_NA := 0;
   BB2_SR_K.ESV_NA := 5;

END_DATA_BLOCK

DATA_BLOCK "DB108_Antriebe_Bef_UV"
{ S7_Optimized_Access := 'FALSE' }
VERSION : 0.1
NON_RETAIN
   STRUCT
      BB_G1 : "T_ANTRIEB_BEF";   // Belebung - Gebläse 1
      BB_G2 : "T_ANTRIEB_BEF";   // Belebung - Gebläse 2
      BB_G3 : "T_ANTRIEB_BEF";   // Belebung - Gebläse 3
      BB_SHL_G1 : "T_ANTRIEB_BEF";   // Belebung - Schallhaubenlüfter Gebläse 1
      BB_SHL_G2 : "T_ANTRIEB_BEF";   // Belebung - Schallhaubenlüfter Gebläse 2
      BB_SHL_G3 : "T_ANTRIEB_BEF";   // Belebung - Schallhaubenlüfter Gebläse 3
      BB_AV : "T_ANTRIEB_BEF";   // Belebung - Gebläsestation - Abluftventilator
      BB_LS1 : "T_ANTRIEB_BEF";   // Belebung - Gebläsestation - Luftwegschieber 1
      BB_LS2 : "T_ANTRIEB_BEF";   // Belebung - Gebläsestation - Luftwegschieber 2
      BB1_RZP1 : "T_ANTRIEB_BEF";   // Becken 1 - Rezipumpe 1
      BB1_RZP2 : "T_ANTRIEB_BEF";   // Becken 1 - Rezipumpe 2
      BB1_UeSP : "T_ANTRIEB_BEF";   // Becken 1 - ÜSS-Pumpe
      BB1_AS1 : "T_ANTRIEB_BEF";   // Becken 1 - Ablaufschieber 1
      BB1_AS2 : "T_ANTRIEB_BEF";   // Becken 1 - Ablaufschieber 2
      BB1_SR1 : "T_ANTRIEB_BEF";   // Becken 1 - MV Schlammrückführung 1
      BB1_SR2 : "T_ANTRIEB_BEF";   // Becken 1 - MV Schlammrückführung 2
      BB2_RZP1 : "T_ANTRIEB_BEF";   // Becken 2 - Rezipumpe 1
      BB2_RZP2 : "T_ANTRIEB_BEF";   // Becken 2 - Rezipumpe 2
      BB2_UeSP : "T_ANTRIEB_BEF";   // Becken 2 - ÜSS-Pumpe
      BB2_AS1 : "T_ANTRIEB_BEF";   // Becken 2 - Ablaufschieber 1
      BB2_AS2 : "T_ANTRIEB_BEF";   // Becken 2 - Ablaufschieber 2
      BB2_SR1 : "T_ANTRIEB_BEF";   // Becken 2 - MV Schlammrückführung 1
      BB2_SR2 : "T_ANTRIEB_BEF";   // Becken 2 - MV Schlammrückführung 2
      BB1_SR_K : "T_ANTRIEB_BEF";   // Becken 1- Druckluftkompressor Schlammrückführung
      Zulauf_AR_P1 : "T_ANTRIEB_BEF";   // Zulauf - Pumpwerk "Alter Rechen" - Pumpe 1
      Zulauf_AR_P2 : "T_ANTRIEB_BEF";   // Zulauf - Pumpwerk "Alter Rechen" - Pumpe 2
      Zulauf_AS : "T_ANTRIEB_BEF";   // Zulauf - Vorlagebehälter - Absperrschieber
      Zulauf_RA_SA : "T_ANTRIEB_BEF";   // Zulauf - Rechen - Sieb
      Zulauf_RA_HZS : "T_ANTRIEB_BEF";   // Zulauf - Rechen - HZS
      Zulauf_RA_VKS : "T_ANTRIEB_BEF";   // Zulauf - Rechen - VZS
      Zulauf_RA_V : "T_ANTRIEB_BEF";   // Zulauf - Rechen - Belüfter
      Zulauf_RA_RP : "T_ANTRIEB_BEF";   // Zulauf - Rechen - Räumpaddel
      Zulauf_RA_FP : "T_ANTRIEB_BEF";   // Zulauf - Rechen - Fettpumpe
      Schlamm_BP : "T_ANTRIEB_BEF";   // Schlamm - Beschickungspumpe Schlammbeete
      Truebwasser_P1 : "T_ANTRIEB_BEF";   // Trübwasserpumpwerk - Pumpe 1
      Truebwasser_P2 : "T_ANTRIEB_BEF";   // Trübwasserpumpwerk - Pumpe 2
      Schlamm_AS : "T_ANTRIEB_BEF";   // Schlamm - Absperrschieber Schlammbeete
      BB2_SR_K : "T_ANTRIEB_BEF";   // Becken 2 - Druckluftkompressor Schlammrückführung
      Zulauf_DosP : "T_ANTRIEB_BEF";   // Zulauf - Dosierpumpe
   END_STRUCT;


